(* IEC 61131-3 sources: smart-home/SmartHome/plc (part 3) *)

(* ---- Tn_ReadSensors.st ---- *)
(****************************************************************************
**
** Copyright (C) 2021 Francesco Mandracci
** Contact: https://github.com/fmandracci/smart-home
**
** This file is part of the Smart Home Framework.
**
** Commercial License Usage
** Licensees holding valid commercial licenses may use this file in
** accordance with the terms contained in a written agreement
** between you and the copyright owner.
**
** GNU Lesser General Public License Usage
** Alternatively, this file may be used under the terms of the GNU Lesser
** General Public License version 3 as published by the Free Software
** Foundation and appearing in the file LICENSE included in the
** packaging of this file. Please review the following information to
** ensure the GNU Lesser General Public License version 3 requirements
** will be met: https://www.gnu.org/licenses/lgpl-3.0.html.
**
****************************************************************************)

FUNCTION Tn_ReadSensors
#import "Crosstable.gvl"
#import "Resource1.gvl"
VAR_INPUT
	n  : UINT; (* Tn                     *)
    ES : INT;  (* PLC_Tn_enabled_sensors *)
END_VAR
VAR_IN_OUT
    T1 : INT;  (* PLC_Tn_temperature     *)
    T2 : INT;  (* PLC_Tn_temperature_bis *)
    T3 : INT;  (* PLC_Tn_temperature_ext *)

    H1 : INT;  (* PLC_Tn_humidity        *)
    H2 : INT;  (* PLC_Tn_humidity_bis    *)
    H3 : INT;  (* PLC_Tn_humidity_ext    *)
END_VAR

	(* INPUT: sensors *)
	if PLC_control_type = ControlType_3 or PLC_control_type = ControlType_4 or PLC_control_type = ControlType_15 then
		(* TPAC1007_04_AD Local I/O AI1..3 on RTU3 *)
		if ES >= 1 then
			if NODE_31_STATUS = NODE_NODE_OK then
				SetAnIn_PT100R(PLC_AnInConf_1, PLC_AnIn1Filter);
				T1 := PLC_AnIn_1;
			else
				T1 := TemperatureErrorValue;
			end_if;
			H1 := 0;
		end_if;
		if ES >= 2 then
			if NODE_31_STATUS = NODE_NODE_OK then
				SetAnIn_PT100R(PLC_AnInConf_2, PLC_AnIn2Filter);
				T2 := PLC_AnIn_2;
			else
				T2 := TemperatureErrorValue;
			end_if;
			H2 := 0;
		end_if;
		if ES >= 3 then
			if NODE_31_STATUS = NODE_NODE_OK then
				SetAnIn_PT100R(PLC_AnInConf_3, PLC_AnIn3Filter);
				T3 := PLC_AnIn_3;
			else
				T3 := TemperatureErrorValue;
			end_if;
			H3 := 0;
		end_if;

	elsif (PLC_control_type = ControlType_13 and n <= 3) then
		(* n=1..3 TPAC1007_04_AD Local I/O AI1..3 on RTU3 *)
		if ES >= 1 then
			if NODE_31_STATUS = NODE_NODE_OK then
				case n of
				1:
					SetAnIn_PT100R(PLC_AnInConf_1, PLC_AnIn1Filter);
					T1 := PLC_AnIn_1;
				2:
					SetAnIn_PT100R(PLC_AnInConf_2, PLC_AnIn2Filter);
					T1 := PLC_AnIn_2;
				3:
					SetAnIn_PT100R(PLC_AnInConf_3, PLC_AnIn3Filter);
					T1 := PLC_AnIn_3;
				else ;
				end_case;
			else
				T1 := TemperatureErrorValue;
			end_if;
			H1 := 0;
		end_if;

	elsif PLC_control_type = ControlType_5 or PLC_control_type = ControlType_8 or PLC_control_type = ControlType_12 then
		(* first, second and third (T,H) sensor on RTU3 *)
		if ES <= -1 then
			if NODE_28_STATUS = NODE_NODE_OK then
				T1 := RTU_temperature;
				H1 := RTU_humidity;
			else
				T1 := TemperatureErrorValue;
				H1 := HumidityErrorValue;
			end_if;
		end_if;
		if ES <= -2 then
			if NODE_29_STATUS = NODE_NODE_OK then
				T2 := RTU_temperature_bis;
				H2 := RTU_humidity_bis;
			else
				T2 := TemperatureErrorValue;
				H2 := HumidityErrorValue;
			end_if;
		end_if;
		if ES <= -3 then
			if NODE_30_STATUS = NODE_NODE_OK then
				T3 := RTU_temperature_bis;
				H3 := RTU_humidity_bis;
			else
				T3 := TemperatureErrorValue;
				H3 := HumidityErrorValue;
			end_if;
		end_if;

	elsif PLC_control_type = ControlType_6 then
		(* MPNC 4xAI4 on RTU0 1=C+6 2=B+7 3=A+8 4=base+5, bis,ext varies *)
		if NODE_27_STATUS = NODE_NODE_OK then
			case n of
			1:
				if MPNC_AnInConf_C <> AnIn_MPNCx4_Pt100R then MPNC_AnInConf_C := AnIn_MPNCx4_Pt100R; end_if;
				T1 := MPNC_AnIn_C_3; (* scala *)
				T2 := MPNC_AnIn_C_1; (* lavanderia *)
				T3 := MPNC_AnIn_C_2; (* cantina *)
			2:
				if MPNC_AnInConf_B <> AnIn_MPNCx4_Pt100R then MPNC_AnInConf_B := AnIn_MPNCx4_Pt100R; end_if;
				T1 := MPNC_AnIn_B_3; (* corridoio *)
				T2 := MPNC_AnIn_B_1; (* cucina *)
				T3 := MPNC_AnIn_B_2; (* soggiorno *)
			3:
				if MPNC_AnInConf_A <> AnIn_MPNCx4_Pt100R then MPNC_AnInConf_A := AnIn_MPNCx4_Pt100R; end_if;
				T1 := MPNC_AnIn_A_3; (* sopra sud *)
				T2 := MPNC_AnIn_A_2; (* sopra nord *)
				T3 := MPNC_AnIn_A_1; (* esterna *)
			4:
				if MPNC_AnInConf_1 <> AnIn_MPNC_Pt100R then MPNC_AnInConf_1 := AnIn_MPNC_Pt100R; end_if;
				if MPNC_AnInConf_2 <> AnIn_MPNC_Pt100R then MPNC_AnInConf_2 := AnIn_MPNC_Pt100R; end_if;
				T1 := MPNC_AnIn_1; (* puffer *)
				T2 := MPNC_AnIn_2; (* ritorno radiatori *)
				T3 := 0;
			else ;
			end_case;
		else
			T1 := TemperatureErrorValue;
			T2 := TemperatureErrorValue;
			T3 := TemperatureErrorValue;
		end_if;
		H1 := 0;
		H2 := 0;
		H3 := 0;

	elsif PLC_control_type = ControlType_14 then
		(* MPNC 4xAI4 on RTU0 1=A 2=B 3=C 4=D _1=t _2=t_bis _3=t_ext *)
		if NODE_27_STATUS = NODE_NODE_OK then
			case n of
			1:
				if MPNC_AnInConf_A <> AnIn_MPNCx4_Pt100R then MPNC_AnInConf_A := AnIn_MPNCx4_Pt100R; end_if;
				T1 := MPNC_AnIn_A_1;
				T2 := MPNC_AnIn_A_2;
				T3 := MPNC_AnIn_A_3;
			2:
				if MPNC_AnInConf_B <> AnIn_MPNCx4_Pt100R then MPNC_AnInConf_B := AnIn_MPNCx4_Pt100R; end_if;
				T1 := MPNC_AnIn_B_1;
				T2 := MPNC_AnIn_B_2;
				T3 := MPNC_AnIn_B_3;
			3:
				if MPNC_AnInConf_C <> AnIn_MPNCx4_Pt100R then MPNC_AnInConf_C := AnIn_MPNCx4_Pt100R; end_if;
				T1 := MPNC_AnIn_C_1;
				T2 := MPNC_AnIn_C_2;
				T3 := MPNC_AnIn_C_3;
			4:
				if MPNC_AnInConf_D <> AnIn_MPNCx4_Pt100R then MPNC_AnInConf_D := AnIn_MPNCx4_Pt100R; end_if;
				T1 := MPNC_AnIn_D_1;
				T2 := MPNC_AnIn_D_2;
				T3 := MPNC_AnIn_D_3;
			else ;
			end_case;
		else
			T1 := TemperatureErrorValue;
			T2 := TemperatureErrorValue;
			T3 := TemperatureErrorValue;
		end_if;
		H1 := 0;
		H2 := 0;
		H3 := 0;

	elsif PLC_control_type = ControlType_7 then
		(* n=1..4 MPNE_C AI1..4 on RTU0; n=5,6 T,H on RTU3 *)
		if n <= 4 then
			if ES >= 1 then
				if NODE_13_STATUS = NODE_NODE_OK then
					case n of
					1:
						SetAnIn_PT100R(MPNE_C_AnIn1Conf, MPNE_C_AnIn1Filter);
						T1 := MPNE_C_AnIn_1;
					2:
						SetAnIn_PT100R(MPNE_C_AnIn2Conf, MPNE_C_AnIn2Filter);
						T1 := MPNE_C_AnIn_2;
					3:
						SetAnIn_PT100R(MPNE_C_AnIn3Conf, MPNE_C_AnIn3Filter);
						T1 := MPNE_C_AnIn_3;
					4:
						SetAnIn_PT100R(MPNE_C_AnIn4Conf, MPNE_C_AnIn4Filter);
						T1 := MPNE_C_AnIn_4;
					else ;
					end_case;
				else
					T1 := TemperatureErrorValue;
				end_if;
				H1 := 0;
			end_if;
		elsif (n = 5) and (ES <= -1) then
			if NODE_28_STATUS = NODE_NODE_OK then
				T1 := RTU_temperature;
				H1 := RTU_humidity;
			else
				T1 := TemperatureErrorValue;
				H1 := HumidityErrorValue;
			end_if;
		elsif (n = 6) and (ES <= -1) then
			if NODE_29_STATUS = NODE_NODE_OK then
				T1 := RTU_temperature_bis;
				H1 := RTU_humidity_bis;
			else
				T1 := TemperatureErrorValue;
				H1 := HumidityErrorValue;
			end_if;
		else
			T1 := TemperatureErrorValue;
			H1 := HumidityErrorValue;
		end_if;

	elsif PLC_control_type = ControlType_10 then
		(* MPNE_C AI1.2 on RTU0 *)
		if ES >= 1 then
			if NODE_13_STATUS = NODE_NODE_OK then
				SetAnIn_PT100R(MPNE_C_AnIn1Conf, MPNE_C_AnIn1Filter);
				T1 := MPNE_C_AnIn_1;
			else
				T1 := TemperatureErrorValue;
			end_if;
			H1 := 0;
		end_if;
		if ES >= 2 then
			if NODE_13_STATUS = NODE_NODE_OK then
				SetAnIn_PT100R(MPNE_C_AnIn2Conf, MPNE_C_AnIn2Filter);
				T2 := MPNE_C_AnIn_2;
			else
				T2 := TemperatureErrorValue;
			end_if;
			H2 := 0;
		end_if;

	elsif PLC_control_type = ControlType_11 then
		(* n=1..4: MPNE_C/D AI(1+2) .. (3+4) on RTU0 *)
		case n of
		1:
			SetAnIn_PT100R(MPNE_C_AnIn1Conf, MPNE_C_AnIn1Filter);
			SetAnIn_PT100R(MPNE_C_AnIn2Conf, MPNE_C_AnIn2Filter);
			T1 := MPNE_C_AnIn_1;
			T2 := MPNE_C_AnIn_2;
		2:
			SetAnIn_PT100R(MPNE_C_AnIn3Conf, MPNE_C_AnIn3Filter);
			SetAnIn_PT100R(MPNE_C_AnIn4Conf, MPNE_C_AnIn4Filter);
			T1 := MPNE_C_AnIn_3;
			T2 := MPNE_C_AnIn_4;
		3:
			SetAnIn_PT100R(MPNE_D_AnIn1Conf, MPNE_D_AnIn1Filter);
			SetAnIn_PT100R(MPNE_D_AnIn2Conf, MPNE_D_AnIn2Filter);
			T1 := MPNE_D_AnIn_1;
			T2 := MPNE_D_AnIn_2;
		4:
			SetAnIn_PT100R(MPNE_D_AnIn3Conf, MPNE_D_AnIn3Filter);
			SetAnIn_PT100R(MPNE_D_AnIn4Conf, MPNE_D_AnIn4Filter);
			T1 := MPNE_D_AnIn_3;
			T2 := MPNE_D_AnIn_4;
		else ;
		end_case;

	end_if;

END_FUNCTION

(* ---- Tn_SetDigOut_lamp.st ---- *)
(****************************************************************************
**
** Copyright (C) 2021 Francesco Mandracci
** Contact: https://github.com/fmandracci/smart-home
**
** This file is part of the Smart Home Framework.
**
** Commercial License Usage
** Licensees holding valid commercial licenses may use this file in
** accordance with the terms contained in a written agreement
** between you and the copyright owner.
**
** GNU Lesser General Public License Usage
** Alternatively, this file may be used under the terms of the GNU Lesser
** General Public License version 3 as published by the Free Software
** Foundation and appearing in the file LICENSE included in the
** packaging of this file. Please review the following information to
** ensure the GNU Lesser General Public License version 3 requirements
** will be met: https://www.gnu.org/licenses/lgpl-3.0.html.
**
****************************************************************************)

FUNCTION Tn_SetDigOut_lamp
#import "Crosstable.gvl"
#import "Resource1.gvl"
VAR_INPUT
    x : UINT;
    value : BOOL;
END_VAR

	if PLC_control_type = ControlType_3 or PLC_control_type = ControlType_4 then
		(* TPAC1007_04_AD Local I/O DO1..5 DI7..11 on RTU3 *)
		case x of
		1: if PLC_DigDir_1 <> DigDir_OUT then PLC_DigDir_1 := DigDir_OUT; end_if;
	       if PLC_DigOut_1 <> value      then PLC_DigOut_1 := value; end_if;
		2: if PLC_DigDir_2 <> DigDir_OUT then PLC_DigDir_2 := DigDir_OUT; end_if;
	       if PLC_DigOut_2 <> value      then PLC_DigOut_2 := value; end_if;
		3: if PLC_DigDir_3 <> DigDir_OUT then PLC_DigDir_3 := DigDir_OUT; end_if;
	       if PLC_DigOut_3 <> value      then PLC_DigOut_3 := value; end_if;
		4: if PLC_DigDir_4 <> DigDir_OUT then PLC_DigDir_4 := DigDir_OUT; end_if;
	       if PLC_DigOut_4 <> value      then PLC_DigOut_4 := value; end_if;
		5: if PLC_DigDir_5 <> DigDir_OUT then PLC_DigDir_5 := DigDir_OUT; end_if;
	       if PLC_DigOut_5 <> value      then PLC_DigOut_5 := value; end_if;
 	    else ;
	    end_case;

	elsif PLC_control_type = ControlType_5 or PLC_control_type = ControlType_8 then
		(* Fast I/O FO5..8 FO5..8 on GPIO *)
		case x of
		1: if PLC_FastIO_5 <> value then PLC_FastIO_5 := value; end_if;
		2: if PLC_FastIO_6 <> value then PLC_FastIO_6 := value; end_if;
		3: if PLC_FastIO_7 <> value then PLC_FastIO_7 := value; end_if;
		4: if PLC_FastIO_8 <> value then PLC_FastIO_8 := value; end_if;
 	    else ;
	    end_case;

	else
		; (* no lamps *)
	end_if;

END_FUNCTION

(* ---- Tn_SetDigOut_thermo.st ---- *)
(****************************************************************************
**
** Copyright (C) 2021 Francesco Mandracci
** Contact: https://github.com/fmandracci/smart-home
**
** This file is part of the Smart Home Framework.
**
** Commercial License Usage
** Licensees holding valid commercial licenses may use this file in
** accordance with the terms contained in a written agreement
** between you and the copyright owner.
**
** GNU Lesser General Public License Usage
** Alternatively, this file may be used under the terms of the GNU Lesser
** General Public License version 3 as published by the Free Software
** Foundation and appearing in the file LICENSE included in the
** packaging of this file. Please review the following information to
** ensure the GNU Lesser General Public License version 3 requirements
** will be met: https://www.gnu.org/licenses/lgpl-3.0.html.
**
****************************************************************************)

FUNCTION Tn_SetDigOut_thermo
#import "Crosstable.gvl"
#import "Resource1.gvl"
VAR_INPUT
    n : UINT;
    heating : BOOL;
	only_mantain: BOOL;
	temperature : INT;
	temperature_bis : INT;
END_VAR
VAR_IN_OUT
	last_R : UINT;
END_VAR

	if PLC_control_type = ControlType_3 then
		(* TPAC1007_04_AD DigOut 6 *)
		if NODE_31_STATUS = NODE_NODE_OK then
	    	if PLC_DigDir_6 <> DigDir_OUT then PLC_DigDir_6 := DigDir_OUT; end_if;
			if only_mantain then
				; (* do nothing *)
			else
		        if PLC_DigOut_6 <> HEATING then PLC_DigOut_6 := HEATING; end_if;
		    end_if;
	    end_if;

	elsif PLC_control_type = ControlType_4 or PLC_control_type = ControlType_5 or PLC_control_type = ControlType_8 then
		(* ARQ01 relè *)
		if NODE_10_STATUS = NODE_NODE_OK then
		    if only_mantain then
				; (* do nothing *)
			else
		        if ARQ_Rele <> HEATING then ARQ_Rele := HEATING; end_if;
			end_if;
		end_if;

	elsif PLC_control_type = ControlType_7 then
		(* n=1..4: MPNE_C DigOut 1..4 *)
		if NODE_13_STATUS = NODE_NODE_OK then
			if only_mantain then
				; (* do nothing *)
			else
	    		case n of
				1:
			    	if MPNE_C_DigDir_1 <> DigDir_OUT then MPNE_C_DigDir_1 := DigDir_OUT; end_if;
			        if MPNE_C_DigOut_1 <> HEATING    then MPNE_C_DigOut_1 := HEATING   ; end_if;
				2:
			    	if MPNE_C_DigDir_2 <> DigDir_OUT then MPNE_C_DigDir_2 := DigDir_OUT; end_if;
			        if MPNE_C_DigOut_2 <> HEATING    then MPNE_C_DigOut_2 := HEATING   ; end_if;
				3:
			    	if MPNE_C_DigDir_3 <> DigDir_OUT then MPNE_C_DigDir_3 := DigDir_OUT; end_if;
			        if MPNE_C_DigOut_3 <> HEATING    then MPNE_C_DigOut_3 := HEATING   ; end_if;
				4:
			    	if MPNE_C_DigDir_4 <> DigDir_OUT then MPNE_C_DigDir_4 := DigDir_OUT; end_if;
			        if MPNE_C_DigOut_4 <> HEATING    then MPNE_C_DigOut_4 := HEATING   ; end_if;
				5:
			    	if MPNE_C_DigDir_5 <> DigDir_OUT then MPNE_C_DigDir_5 := DigDir_OUT; end_if;
			        if MPNE_C_DigOut_5 <> HEATING    then MPNE_C_DigOut_5 := HEATING   ; end_if;
				6:
			    	if MPNE_C_DigDir_6 <> DigDir_OUT then MPNE_C_DigDir_6 := DigDir_OUT; end_if;
			        if MPNE_C_DigOut_6 <> HEATING    then MPNE_C_DigOut_6 := HEATING   ; end_if;
				else ;
				end_case;
			end_if;
		end_if;

	elsif PLC_control_type = ControlType_10 then
		(* MPNE_C DigOut 1 *)
		if NODE_13_STATUS = NODE_NODE_OK then
	    	if MPNE_C_DigDir_1 <> DigDir_OUT then MPNE_C_DigDir_1 := DigDir_OUT; end_if;

			if only_mantain then
				; (* do nothing *)
			else
		        if heating then (* see also Tn_OverHeat() *)
			    	if not MPNE_C_DigOut_1 then MPNE_C_DigOut_1 := true; end_if;
				else
			    	if MPNE_C_DigOut_1 then MPNE_C_DigOut_1 := false; end_if;
				end_if;
			end_if;
		end_if;

	elsif PLC_control_type = ControlType_11 then
		(* i=1..4: MPNE_C/_D DigOut 1.2 *)
		if n <= 2 then
			if NODE_13_STATUS = NODE_NODE_OK then
				if only_mantain then
					; (* do nothing *)
				else
					case n of
					1:
				    	if MPNE_C_DigDir_1 <> DigDir_OUT then MPNE_C_DigDir_1 := DigDir_OUT; end_if;
						if only_mantain then
							; (* do nothing *)
						else
					        if heating then (* see also Tn_OverHeat() *)
						    	if not MPNE_C_DigOut_1 then MPNE_C_DigOut_1 := true; end_if;
							else
						    	if MPNE_C_DigOut_1 then MPNE_C_DigOut_1 := false; end_if;
							end_if;
						end_if;
					2:
				    	if MPNE_C_DigDir_2 <> DigDir_OUT then MPNE_C_DigDir_2 := DigDir_OUT; end_if;
						if only_mantain then
							; (* do nothing *)
						else
					        if heating then (* see also Tn_OverHeat() *)
						    	if not MPNE_C_DigOut_2 then MPNE_C_DigOut_2 := true; end_if;
							else
						    	if MPNE_C_DigOut_2 then MPNE_C_DigOut_2 := false; end_if;
							end_if;
						end_if;
					else ;
					end_case;
				end_if;
			end_if;
		else
			if NODE_14_STATUS = NODE_NODE_OK then
				if only_mantain then
					; (* do nothing *)
				else
					case n of
					3:
				    	if MPNE_D_DigDir_1 <> DigDir_OUT then MPNE_D_DigDir_1 := DigDir_OUT; end_if;
						if only_mantain then
							; (* do nothing *)
						else
					        if heating then (* see also Tn_OverHeat() *)
						    	if not MPNE_D_DigOut_1 then MPNE_D_DigOut_1 := true; end_if;
							else
						    	if MPNE_D_DigOut_1 then MPNE_D_DigOut_1 := false; end_if;
							end_if;
						end_if;
					4:
				    	if MPNE_D_DigDir_2 <> DigDir_OUT then MPNE_D_DigDir_2 := DigDir_OUT; end_if;
						if only_mantain then
							; (* do nothing *)
						else
					        if heating then (* see also Tn_OverHeat() *)
						    	if not MPNE_D_DigOut_2 then MPNE_D_DigOut_2 := true; end_if;
							else
						    	if MPNE_D_DigOut_2 then MPNE_D_DigOut_2 := false; end_if;
							end_if;
						end_if;
					else ;
					end_case;
				end_if;
			end_if;
		end_if;

	elsif PLC_control_type = ControlType_12 then
		(* FastI/O FO 8 *)
        if only_mantain then
			; (* do nothing *)
		else
	        if PLC_FastIO_8 <> HEATING then PLC_FastIO_8 := HEATING; end_if;
		end_if;

	elsif PLC_control_type = ControlType_13 then
		(* n=1..4: TPAC1007_04_AD DigOut_1..4 *)
		if NODE_31_STATUS = NODE_NODE_OK then
			if only_mantain then
				; (* do nothing *)
			else
		        case n of
				1:
			    	if PLC_DigDir_1 <> DigDir_OUT then PLC_DigDir_1 := DigDir_OUT; end_if;
			        if PLC_DigOut_1 <> HEATING    then PLC_DigOut_1 := HEATING   ; end_if;
				2:
			    	if PLC_DigDir_2 <> DigDir_OUT then PLC_DigDir_2 := DigDir_OUT; end_if;
			        if PLC_DigOut_2 <> HEATING    then PLC_DigOut_2 := HEATING   ; end_if;
				3:
			    	if PLC_DigDir_3 <> DigDir_OUT then PLC_DigDir_3 := DigDir_OUT; end_if;
			        if PLC_DigOut_3 <> HEATING    then PLC_DigOut_3 := HEATING   ; end_if;
				4:
			    	if PLC_DigDir_4 <> DigDir_OUT then PLC_DigDir_4 := DigDir_OUT; end_if;
			        if PLC_DigOut_4 <> HEATING    then PLC_DigOut_4 := HEATING   ; end_if;
				else ;
				end_case;
			end_if;
		end_if;

	elsif PLC_control_type = ControlType_6 then
		(* MPNC 4xAI4 on RTU0 1=C+6 2=B+7 3=A+8 4=base+5, bis,ext varies *)
		if NODE_27_STATUS = NODE_NODE_OK then
			if only_mantain then
				; (* do nothing *)
			else
		        case n of
				1:
			    	if MPNC_DigDir_6 <> DigDir_OUT then MPNC_DigDir_6 := DigDir_OUT; end_if;
			        if MPNC_DigOut_6 <> HEATING    then MPNC_DigOut_6 := HEATING   ; end_if;
				2:
			    	if MPNC_DigDir_7 <> DigDir_OUT then MPNC_DigDir_7 := DigDir_OUT; end_if;
			        if MPNC_DigOut_7 <> HEATING    then MPNC_DigOut_7 := HEATING   ; end_if;
				3:
			    	if MPNC_DigDir_8 <> DigDir_OUT then MPNC_DigDir_8 := DigDir_OUT; end_if;
			        if MPNC_DigOut_8 <> HEATING    then MPNC_DigOut_8 := HEATING   ; end_if;
				4:
			    	if MPNC_DigDir_5 <> DigDir_OUT then MPNC_DigDir_5 := DigDir_OUT; end_if;
			        if MPNC_DigOut_5 <> HEATING    then MPNC_DigOut_5 := HEATING   ; end_if;
				else ;
				end_case;
			end_if;
		end_if;

	elsif PLC_control_type = ControlType_14 then
		(* n=1..4: MPNC base DigOut_1..4 *)
		if NODE_27_STATUS = NODE_NODE_OK then
			if only_mantain then
				; (* do nothing *)
			else
		        case n of
				1:
			    	if MPNC_DigDir_1 <> DigDir_OUT then MPNC_DigDir_1 := DigDir_OUT; end_if;
			        if MPNC_DigOut_1 <> HEATING    then MPNC_DigOut_1 := HEATING   ; end_if;
				2:
			    	if MPNC_DigDir_2 <> DigDir_OUT then MPNC_DigDir_2 := DigDir_OUT; end_if;
			        if MPNC_DigOut_2 <> HEATING    then MPNC_DigOut_2 := HEATING   ; end_if;
				3:
			    	if MPNC_DigDir_3 <> DigDir_OUT then MPNC_DigDir_3 := DigDir_OUT; end_if;
			        if MPNC_DigOut_3 <> HEATING    then MPNC_DigOut_3 := HEATING   ; end_if;
				4:
			    	if MPNC_DigDir_4 <> DigDir_OUT then MPNC_DigDir_4 := DigDir_OUT; end_if;
			        if MPNC_DigOut_4 <> HEATING    then MPNC_DigOut_4 := HEATING   ; end_if;
				else ;
				end_case;
		    end_if;
	    end_if;

	elsif PLC_control_type = ControlType_15 then
		(* TPAC1007_04_AD DigOut_8 *)
		if NODE_31_STATUS = NODE_NODE_OK then
	    	if PLC_DigDir_8 <> DigDir_OUT then PLC_DigDir_8 := DigDir_OUT; end_if;
	        if only_mantain then
				; (* do nothing *)
			else
		        if PLC_DigOut_8 <> HEATING then PLC_DigOut_8 := HEATING; end_if;
			end_if;
	    end_if;

	end_if;

END_FUNCTION

(* ---- Tn_Watchdog.st ---- *)
(****************************************************************************
**
** Copyright (C) 2021 Francesco Mandracci
** Contact: https://github.com/fmandracci/smart-home
**
** This file is part of the Smart Home Framework.
**
** Commercial License Usage
** Licensees holding valid commercial licenses may use this file in
** accordance with the terms contained in a written agreement
** between you and the copyright owner.
**
** GNU Lesser General Public License Usage
** Alternatively, this file may be used under the terms of the GNU Lesser
** General Public License version 3 as published by the Free Software
** Foundation and appearing in the file LICENSE included in the
** packaging of this file. Please review the following information to
** ensure the GNU Lesser General Public License version 3 requirements
** will be met: https://www.gnu.org/licenses/lgpl-3.0.html.
**
****************************************************************************)

FUNCTION Tn_Watchdog
#import "Crosstable.gvl"
#import "Resource1.gvl"

	if (PLC_control_type = ControlType_4) or (PLC_control_type = ControlType_5) or (PLC_control_type = ControlType_8) then
		if ARQ_Watchdog <> WatchDogTimeout_s and NODE_10_STATUS = NODE_NODE_OK then
			ARQ_Watchdog := WatchDogTimeout_s;
		end_if;
	end_if;

END_FUNCTION

(* ---- FilteredSensors.st ---- *)
(****************************************************************************
**
** Copyright (C) 2021 Francesco Mandracci
** Contact: https://github.com/fmandracci/smart-home
**
** This file is part of the Smart Home Framework.
**
** Commercial License Usage
** Licensees holding valid commercial licenses may use this file in
** accordance with the terms contained in a written agreement
** between you and the copyright owner.
**
** GNU Lesser General Public License Usage
** Alternatively, this file may be used under the terms of the GNU Lesser
** General Public License version 3 as published by the Free Software
** Foundation and appearing in the file LICENSE included in the
** packaging of this file. Please review the following information to
** ensure the GNU Lesser General Public License version 3 requirements
** will be met: https://www.gnu.org/licenses/lgpl-3.0.html.
**
****************************************************************************)

FUNCTION_BLOCK FilteredSensors
#import "Crosstable.gvl"
#import "Resource1.gvl"
VAR_INPUT
	n  : UINT; (* Tn                     *)
    ES : INT;  (* PLC_Tn_enabled_sensors *)
END_VAR
VAR_IN_OUT
    T1 : INT;  (* PLC_Tn_temperature     *)
    T2 : INT;  (* PLC_Tn_temperature_bis *)
    T3 : INT;  (* PLC_Tn_temperature_ext *)

    H1 : INT;  (* PLC_Tn_humidity        *)
    H2 : INT;  (* PLC_Tn_humidity_bis    *)
    H3 : INT;  (* PLC_Tn_humidity_ext    *)
END_VAR
VAR
    T1_value : INT := TemperatureErrorValue;
    T2_value : INT := TemperatureErrorValue;
    T3_value : INT := TemperatureErrorValue;
	i : INT;
	s : INT;
	m : INT;
	first_time : BOOL := true;
	T1_array : array [1 .. RollingAverageSize] of INT;
	T2_array : array [1 .. RollingAverageSize] of INT;
	T3_array : array [1 .. RollingAverageSize] of INT;
END_VAR

	if first_time then
		first_time := false;
		for i := 1 to RollingAverageSize by 1 do
			T1_array[i] := TemperatureErrorValue;
			T2_array[i] := TemperatureErrorValue;
			T3_array[i] := TemperatureErrorValue;
		end_for;
	end_if;

    Tn_ReadSensors(n, ES, T1_value, T2_value, T3_value, H1, H2, H3);

	if (abs(ES) >= 1) and (T1_value <> TemperatureErrorValue) then
		s := 0;
		for i := 1 to (RollingAverageSize - 1) by 1 do
			T1_array[i] := T1_array[i + 1];
			s := s + T1_array[i];
		end_for;
		T1_array[RollingAverageSize] := T1_value;
		s := s + T1_value;
		m := s / RollingAverageSize;
		if (s mod RollingAverageSize) >= HalfRollingAverageSize then
			m := m + 1;
		end_if;
		if abs(T1_value - m) <= RollingAverageMaxDeltaT then
			T1 := m;
		else
			for i := 1 to RollingAverageSize by 1 do
				T1_array[i] := T1_value;
			end_for;
			T1 := T1_value;
		end_if;
	else
		T1 := TemperatureErrorValue;
	end_if;

	if (abs(ES) >= 2) and (T2_value <> TemperatureErrorValue) then
		s := 0;
		for i := 1 to (RollingAverageSize - 1) by 1 do
			T2_array[i] := T2_array[i + 1];
			s := s + T2_array[i];
		end_for;
		T2_array[RollingAverageSize] := T2_value;
		s := s + T2_value;
		m := s / RollingAverageSize;
		if (s mod RollingAverageSize) >= HalfRollingAverageSize then
			m := m + 1;
		end_if;
		if abs(T2_value - m) <= RollingAverageMaxDeltaT then
			T2 := m;
		else
			for i := 1 to RollingAverageSize by 1 do
				T2_array[i] := T2_value;
			end_for;
			T2 := T2_value;
		end_if;
	else
		T2 := TemperatureErrorValue;
	end_if;

	if (abs(ES) >= 3) and (T3_value <> TemperatureErrorValue) then
		s := 0;
		for i := 1 to (RollingAverageSize - 1) by 1 do
			T3_array[i] := T3_array[i + 1];
			s := s + T3_array[i];
		end_for;
		T3_array[RollingAverageSize] := T3_value;
		s := s + T3_value;
		m := s / RollingAverageSize;
		if (s mod RollingAverageSize) >= HalfRollingAverageSize then
			m := m + 1;
		end_if;
		if abs(T3_value - m) <= RollingAverageMaxDeltaT then
			T3 := m;
		else
			for i := 1 to RollingAverageSize by 1 do
				T3_array[i] := T3_value;
			end_for;
			T3 := T3_value;
		end_if;
	else
		T3 := TemperatureErrorValue;
	end_if;

END_FUNCTION_BLOCK

(* ---- LampImpulse.st ---- *)
(****************************************************************************
**
** Copyright (C) 2021 Francesco Mandracci
** Contact: https://github.com/fmandracci/smart-home
**
** This file is part of the Smart Home Framework.
**
** Commercial License Usage
** Licensees holding valid commercial licenses may use this file in
** accordance with the terms contained in a written agreement
** between you and the copyright owner.
**
** GNU Lesser General Public License Usage
** Alternatively, this file may be used under the terms of the GNU Lesser
** General Public License version 3 as published by the Free Software
** Foundation and appearing in the file LICENSE included in the
** packaging of this file. Please review the following information to
** ensure the GNU Lesser General Public License version 3 requirements
** will be met: https://www.gnu.org/licenses/lgpl-3.0.html.
**
****************************************************************************)

FUNCTION_BLOCK LampImpulse
VAR_INPUT
    x  : UINT;
END_VAR
VAR_IN_OUT
    PLC_Tn_lamp_x : BOOL;
    SRV_Tn_lamp_x : BOOL;
    PLC_Tn_lamp_feedback_x : BOOL;
END_VAR
VAR
	active : BOOL := false;
END_VAR;

	if active then
        Tn_SetDigOut_lamp(x, false);
		PLC_Tn_lamp_x := false;
        SRV_Tn_lamp_x := false;
		active := false;
    else
	    if PLC_Tn_lamp_x or SRV_Tn_lamp_x then
	        Tn_SetDigOut_lamp(x, true);
			active := true;
		end_if;
	end_if;

    PLC_Tn_lamp_feedback_x := Tn_GetDigIn_lamp(x);

END_FUNCTION_BLOCK

(* ---- Thermostat.st ---- *)
(****************************************************************************
**
** Copyright (C) 2021 Francesco Mandracci
** Contact: https://github.com/fmandracci/smart-home
**
** This file is part of the Smart Home Framework.
**
** Commercial License Usage
** Licensees holding valid commercial licenses may use this file in
** accordance with the terms contained in a written agreement
** between you and the copyright owner.
**
** GNU Lesser General Public License Usage
** Alternatively, this file may be used under the terms of the GNU Lesser
** General Public License version 3 as published by the Free Software
** Foundation and appearing in the file LICENSE included in the
** packaging of this file. Please review the following information to
** ensure the GNU Lesser General Public License version 3 requirements
** will be met: https://www.gnu.org/licenses/lgpl-3.0.html.
**
****************************************************************************)

FUNCTION_BLOCK Thermostat
#import "Crosstable.gvl"
#import "Resource1.gvl"
VAR_INPUT
	N : UINT;   (* Tn                             *)
    ES : INT;   (* PLC_Tn_enabled_sensors         *)
	NT : BOOL;  (* PLC_Tn_nighttime               *)

    T_1 : INT;  (* PLC_Tn_temperature             *)
    T_2 : INT;  (* PLC_Tn_temperature_bis         *)

    H_1 : INT;  (* PLC_Tn_humidity                *)
    H_2 : INT;  (* PLC_Tn_humidity_bis            *)

	M_W : UINT; (* PLC_Tn_max_request_W           *)
	A_W : UINT; (* PLC_EP_Tn_assigned_W           *)
END_VAR
VAR_IN_OUT
	PRW : UINT; (* PLC_Tn_requested_W             *)
	SRW : UINT; (* SRV_Tn_requested_W             *)

    TSP : INT;  (* PLC_Tn_temperature_setpoint    *)
    TSPN: INT;  (* PLC_Tn_temperature_setpoint_nt *)

    HSP : INT;  (* PLC_Tn_humidity_setpoint       *)
    HSPN: INT;  (* PLC_Tn_humidity_setpoint_nt    *)

    PLC_STATUS  : INT ; (* PLC_Tn_heating_status  *)
    PLC_TIMER   : INT ; (* PLC_Tn_heating_timer   *)
    PLC_HEATING : BOOL; (* PLC_Tn_heating         *)

    SRV_STATUS  : INT ; (* SRV_Tn_heating_status  *)
    SRV_TIMER   : INT ; (* SRV_Tn_heating_timer   *)
    SRV_HEATING : BOOL; (* SRV_Tn_heating         *)

    DH  : UDINT ; (* PLC_Tn_daily_heating_s       *)
    MH  : UDINT ; (* PLC_Tn_monthly_heating_s     *)
END_VAR
VAR
	HEATING : BOOL;
	TIMER : INT;
	STATUS : INT;
	A_TSP : INT; (* actual temperature setpoint, changed by ECONOMY, COMFORT, BOOST and nightime *)
	A_HSP : INT; (* actual humidity setpoint, NOT changed by ECONOMY, COMFORT, BOOST and nightime *)
	last_R : UINT := 0;
END_VAR;

	STATUS := PLC_STATUS;
	TIMER := PLC_TIMER;
	HEATING := PLC_HEATING;

	(* ----------------- 1/4 common ----------------- *)

	(* check nightime and limits *)
	if NT then
		A_TSP := Tn_CheckSetpoint_T(TSPN);
		A_HSP := Tn_CheckSetpoint_H(HSPN);
		(* NB: may change setpoints <---------------- *)
		if TSPN <> A_TSP then TSPN := A_TSP; end_if;
		if HSPN <> A_HSP then HSPN := A_HSP; end_if;
	else
		A_TSP := Tn_CheckSetpoint_T(TSP);
		A_HSP := Tn_CheckSetpoint_H(HSP);
		(* NB: may change setpoints <---------------- *)
		if TSP <> A_TSP then TSP := A_TSP; end_if;
		if HSP <> A_HSP then HSP := A_HSP; end_if;
	end_if;

	(* check timer *)
	if STATUS > HEATING_AUTO then
		if TIMER > 0 then
		    TIMER := TIMER - 1;
		else
			STATUS := HEATING_AUTO;
			TIMER := 0;
		end_if;
	end_if;

	(* check special states *)
	case STATUS of
	HEATING_AUTO:
		A_TSP := A_TSP;
	HEATING_ECONOMY:
		A_TSP := A_TSP - 20; (* -2°C*) (* ex: -10% A_TSP - (A_TSP * 100) / 10; *)
	HEATING_COMFORT:
		A_TSP := A_TSP + 20; (* +2°C*) (* ex: +10% A_TSP + (A_TSP * 100) / 10; *)
	HEATING_BOOST:
		A_TSP := TemperatureSetPoint_max;
	else
		;
	end_case;

	(* check limits after changes *)
	A_TSP := Tn_CheckSetpoint_T(A_TSP);
	A_HSP := Tn_CheckSetpoint_H(A_HSP);

	(* ----------------- 2/4 common control ----------------- *)

	if PLC_control_type = ControlType_0 or PLC_control_type = ControlType_1  or PLC_control_type = ControlType_2 then
		(* no thermostat *)
	    HEATING := false;

	elsif ES = 0 or (abs(ES) >= 1 and T_1 = TemperatureErrorValue) or (abs(ES) >= 2 and T_2 = TemperatureErrorValue) then
		(* sensor read error *)
	    HEATING := false;

	elsif (ES <= -1 and H_1 = HumidityErrorValue) or (ES <= -2 and H_2 = HumidityErrorValue) then
		(* sensor read error *)
	    HEATING := false;

	elsif (PLC_control_type = ControlType_6 and n = 4) or (PLC_control_type = ControlType_15 and n = 1) then
		(* differential thermostat (puffer) *)
		if PLC_UPTIME_s <= 25 then
			(* waiting for sensors settling *)
			HEATING := false;
		elsif STATUS >= HEATING_AUTO then
			(* heating enabled *)
			if HEATING then
				(* heating was ON *)
				if T_1 < (T_2 - TemperatureHysteresis) then
					(* puffer is colder than thermo water *)
					HEATING := false;
				end_if;
			else
				(* heating was off *)
				if  T_1 >= (T_2 + TemperatureHysteresis) then
					(* puffer is warmer than thermo water *)
					HEATING := true;
				end_if;
			end_if;
		else
			HEATING := false;
			TIMER := 0;
		end_if;

	else
		(* standard thermostat *)
		if PLC_UPTIME_s <= 25 then
			(* waiting for sensors settling *)
			HEATING := false;
		elsif STATUS >= HEATING_AUTO then
			(* heating enabled *)
			if HEATING then
				(* heating was ON *)
				if (ES <= -2)   and ( T_1 >= (A_TSP + TemperatureHysteresis) AND T_2 >= (A_TSP + TemperatureHysteresis) AND H_1 <= (A_HSP - HumidityHysteresis) AND H_2 <= (A_HSP - HumidityHysteresis) ) then
					(* two T,H sensors *)
					HEATING := false;
				elsif (ES = -1) and ( T_1 >= (A_TSP + TemperatureHysteresis)                                            AND H_1 <= (A_HSP - HumidityHysteresis)                                     ) then
					(* one T,H sensor *)
					HEATING := false;
				elsif (ES = 0) then
					(* nothing *)
					HEATING := false;
				elsif (ES = 1)  and ( T_1 >= (A_TSP + TemperatureHysteresis) ) then
					(* one Pt100 *)
					HEATING := false;
				elsif (ES >= 2) and ( T_1 >= (A_TSP + TemperatureHysteresis) AND T_2 >= (A_TSP + TemperatureHysteresis)  ) then
					(* two Pt100s *)
					HEATING := false;
				end_if;
			else
				(* heating was off *)
				if (ES <= -2)   and ( T_1 <= (A_TSP - TemperatureHysteresis) OR T_2 <= (A_TSP - TemperatureHysteresis) OR H_1 >= (A_HSP + HumidityHysteresis) OR H_2 >= (A_HSP + HumidityHysteresis) ) then
					(* two T,H sensors *)
					HEATING := true;
				elsif (ES = -1) and ( T_1 <= (A_TSP - TemperatureHysteresis)                                           OR H_1 >= (A_HSP + HumidityHysteresis)                                    ) then
					(* one T,H sensor *)
					HEATING := true;
				elsif (ES = 0) then
					(* nothing *)
					HEATING := false;
				elsif (ES = 1)  and ( T_1 <= (A_TSP - TemperatureHysteresis) ) then
					(* one Pt100 *)
					HEATING := true;
				elsif (ES >= 2) and ( T_1 <= (A_TSP - TemperatureHysteresis) OR T_2 <= (A_TSP - TemperatureHysteresis) ) then
					(* two Pt100s *)
					HEATING := true;
				end_if;
			end_if;
		else
			HEATING := false;
			TIMER := 0;
		end_if;

	end_if;

	(* ----------------- 3/4 specific control and action ----------------- *)

	if HEATING and Tn_OverHeat(n, T_1, T_2) then
		HEATING := false;
	end_if;

	if M_W = 0 or not PLC_EP_exists then
		(* no load balancing *)
	   	Tn_SetDigOut_thermo(n, HEATING, false, T_1, T_2, last_R);
		if PRW <> 0 then
			PRW := 0; (* PLC_Tn_requested_W := 0 *)
		end_if;

	elsif not PLC_EP_isOK then
		(* safe state *)
		HEATING := false;
	   	Tn_SetDigOut_thermo(n, false, false, T_1, T_2, last_R);

	elsif not HEATING then
		(* simply power off *)
	   	Tn_SetDigOut_thermo(n, false, false, T_1, T_2, last_R);
		PRW := 0; (* PLC_Tn_requested_W *)
		if SRW <> 0 then SRW := 0; end_if; (* SRV_Tn_requested_W *)

	else

		case PLC_EP_tic_in_tac of

	    0: (* request time *)
			PRW := M_W; (* PLC_Tn_requested_W := PLC_Tn_max_request_W *)
			if SRW <> M_W then
				SRW := M_W; (* SRV_Tn_requested_W := PLC_Tn_max_request_W *)
			end_if;
			(* wait, only maintain the current status *)
			Tn_SetDigOut_thermo(n, false, true, T_1, T_2, last_R);

		1: (* transmission time *)
			(* wait, only maintain the current status *)
			Tn_SetDigOut_thermo(n, false, true, T_1, T_2, last_R);

		Decision_TicInTac: (* decision time *)
			(* wait, only maintain the current status *)
			Tn_SetDigOut_thermo(n, false, true, T_1, T_2, last_R);

		3: (* transmission time *)
			(* wait, only maintain the current status *)
			Tn_SetDigOut_thermo(n, false, true, T_1, T_2, last_R);

		4:	(* power off time *)
			if A_W >= M_W then (* PLC_EP_Tn_assigned_W >= PLC_Tn_max_request_W *)
				(* wait, only maintain the current status *)
				Tn_SetDigOut_thermo(n, false, true, T_1, T_2, last_R);
			else
				(* power off *)
			   	Tn_SetDigOut_thermo(n, false, false, T_1, T_2, last_R);
			end_if;

		5:
			(* action time *)
			if A_W >= M_W then (* PLC_EP_Tn_assigned_W >= PLC_Tn_max_request_W *)
			   	Tn_SetDigOut_thermo(n, true, false, T_1, T_2, last_R);
			else
			   	Tn_SetDigOut_thermo(n, false, false, T_1, T_2, last_R);
			end_if;

		6:
			(* action time bis *)
			if A_W >= M_W then (* PLC_EP_Tn_assigned_W >= PLC_Tn_max_request_W *)
			   	Tn_SetDigOut_thermo(n, true, false, T_1, T_2, last_R);
			else
			   	Tn_SetDigOut_thermo(n, false, false, T_1, T_2, last_R);
			end_if;

		end_case;

	end_if;

	(* ----------------- 4/4 update ----------------- *)

	if PLC_STATUS <> STATUS then
		PLC_STATUS := STATUS;
		SRV_STATUS := STATUS;
	end_if;
	if PLC_TIMER <> TIMER then
		PLC_TIMER := TIMER;
		SRV_TIMER := TIMER;
	end_if;
	if PLC_HEATING <> HEATING then
		PLC_HEATING := HEATING;
		SRV_HEATING := HEATING;
	end_if;

	if (PLC_Hours = 0) and (PLC_Minutes = 0) and (PLC_Seconds = 0) then
		DH := 0;
		if PLC_Day = 1 then
			MH := 0;
		end_if;
	elsif HEATING then
		DH := DH + 1;
		MH := MH + 1;
	end_if;

END_FUNCTION_BLOCK

(* ---- Alarms.st ---- *)
(****************************************************************************
**
** Copyright (C) 2021 Francesco Mandracci
** Contact: https://github.com/fmandracci/smart-home
**
** This file is part of the Smart Home Framework.
**
** Commercial License Usage
** Licensees holding valid commercial licenses may use this file in
** accordance with the terms contained in a written agreement
** between you and the copyright owner.
**
** GNU Lesser General Public License Usage
** Alternatively, this file may be used under the terms of the GNU Lesser
** General Public License version 3 as published by the Free Software
** Foundation and appearing in the file LICENSE included in the
** packaging of this file. Please review the following information to
** ensure the GNU Lesser General Public License version 3 requirements
** will be met: https://www.gnu.org/licenses/lgpl-3.0.html.
**
****************************************************************************)

PROGRAM Alarms
#import "Crosstable.gvl"
#import "Resource1.gvl"
VAR

END_VAR

;

END_PROGRAM

(* ---- BA_main.st ---- *)
(****************************************************************************
**
** Copyright (C) 2021 Francesco Mandracci
** Contact: https://github.com/fmandracci/smart-home
**
** This file is part of the Smart Home Framework.
**
** Commercial License Usage
** Licensees holding valid commercial licenses may use this file in
** accordance with the terms contained in a written agreement
** between you and the copyright owner.
**
** GNU Lesser General Public License Usage
** Alternatively, this file may be used under the terms of the GNU Lesser
** General Public License version 3 as published by the Free Software
** Foundation and appearing in the file LICENSE included in the
** packaging of this file. Please review the following information to
** ensure the GNU Lesser General Public License version 3 requirements
** will be met: https://www.gnu.org/licenses/lgpl-3.0.html.
**
****************************************************************************)

PROGRAM BA_main
#import "Crosstable.gvl"
#import "Resource1.gvl"
VAR
	substatus : UINT := 0;
	timer : TON;
	NEXT_STATUS : UINT := 0;
	NEXT_INDEX : UINT := 0;
END_VAR;

    if not PLC_Iam_BA then
		return;
    end_if;
	if PLC_BA_just_started then
		PLC_BA_just_started := false;
		timer(IN := FALSE);
		substatus := 0;
	end_if;

	BA_Watchdog();

	NEXT_STATUS := PLC_BA_status;
	NEXT_INDEX := PLC_BA_config_index;

	case substatus of

	0: (* ----- recover config  ------------------------------------------- *)

		case PLC_BA_status of
		ALARM_STATUS_ZERO:
			NEXT_INDEX := ALARM_INDEX_NOTHING;
			NEXT_STATUS := ALARM_STATUS_OFF;
		ALARM_STATUS_OFF:
			NEXT_INDEX := ALARM_INDEX_NOTHING;
		ALARM_STATUS_ARMED:
			;
		ALARM_STATUS_ENABLED:
			;
		ALARM_STATUS_RINGING:
			;
		ALARM_STATUS_MUTED:
			;
		ALARM_STATUS_TESTING:
			;
		else
			NEXT_INDEX := ALARM_INDEX_NOTHING;
			NEXT_STATUS := ALARM_STATUS_OFF;
		end_case;

		BA_WriteConfig(NEXT_INDEX, PLC_BA_config_index, PLC_BA_config_mask);
	    PLC_BA_command := ALARM_COMMAND_NONE;
		substatus := 1;

	1: (* ----- waiting config after write -------------------------------- *)

		timer(IN := TRUE, PT := ControlPeriod);
		if timer.Q then
			timer(IN := FALSE);
			substatus := 2;
		end_if;

	2: (* ----- read sensors ---------------------------------------------- *)

		BA_ReadSensors();
		substatus := 3;

	3: (* ----- check sensors --------------------------------------------- *)

		case PLC_BA_status of

		ALARM_STATUS_ZERO:
			BA_ClearOKs();
			NEXT_INDEX := ALARM_INDEX_NOTHING;
			NEXT_STATUS := ALARM_STATUS_OFF;
			BA_WriteConfig(NEXT_INDEX, PLC_BA_config_index, PLC_BA_config_mask);
			substatus := 1;

		ALARM_STATUS_OFF:
			BA_ClearOKs();
			if PLC_BA_command = ALARM_COMMAND_DAYTIME then
				NEXT_STATUS := ALARM_STATUS_ARMED;
				NEXT_INDEX := ALARM_INDEX_DAYTIME;
				BA_WriteConfig(NEXT_INDEX, PLC_BA_config_index, PLC_BA_config_mask);
				substatus := 1;
			elsif PLC_BA_command = ALARM_COMMAND_NIGHTTIME then
				NEXT_STATUS := ALARM_STATUS_ARMED;
				NEXT_INDEX := ALARM_INDEX_NIGHTTIME;
				BA_WriteConfig(NEXT_INDEX, PLC_BA_config_index, PLC_BA_config_mask);
				substatus := 1;
			elsif PLC_BA_command = ALARM_COMMAND_EVERYTHING then
				NEXT_STATUS := ALARM_STATUS_ARMED;
				NEXT_INDEX := ALARM_INDEX_EVERYTHING;
				BA_WriteConfig(NEXT_INDEX, PLC_BA_config_index, PLC_BA_config_mask);
				substatus := 1;
			elsif PLC_BA_command = ALARM_COMMAND_TEST then
				NEXT_STATUS := ALARM_STATUS_TESTING;
				(* NEXT_INDEX := ALARM_INDEX_NOTHING; *)
			 	(* no BA_WriteConfig(NEXT_INDEX, PLC_BA_config_index, PLC_BA_config_mask);     *)
				substatus := 2;
			else
				substatus := 2;
			end_if;

		ALARM_STATUS_ARMED:
			if PLC_BA_command = ALARM_COMMAND_DAYTIME then
				NEXT_INDEX := ALARM_INDEX_DAYTIME;
				BA_WriteConfig(NEXT_INDEX, PLC_BA_config_index, PLC_BA_config_mask);
				substatus := 1;
			elsif PLC_BA_command = ALARM_COMMAND_NIGHTTIME then
				NEXT_INDEX := ALARM_INDEX_NIGHTTIME;
				BA_WriteConfig(NEXT_INDEX, PLC_BA_config_index, PLC_BA_config_mask);
				substatus := 1;
			elsif PLC_BA_command = ALARM_COMMAND_EVERYTHING then
				NEXT_INDEX := ALARM_INDEX_EVERYTHING;
				BA_WriteConfig(NEXT_INDEX, PLC_BA_config_index, PLC_BA_config_mask);
				substatus := 1;
			elsif PLC_BA_command = ALARM_COMMAND_DISABLE then
				NEXT_STATUS := ALARM_STATUS_OFF;
				NEXT_INDEX := ALARM_INDEX_NOTHING;
				BA_WriteConfig(NEXT_INDEX, PLC_BA_config_index, PLC_BA_config_mask);
				substatus := 1;
			elsif PLC_BA_command = ALARM_COMMAND_ENABLE then
				NEXT_STATUS := ALARM_STATUS_ENABLED;
				substatus := 2;
			elsif PLC_BA_command = ALARM_COMMAND_TEST then
				NEXT_STATUS := ALARM_STATUS_TESTING;
				substatus := 2;
			elsif BA_CheckSensors(PLC_BA_config_index) then
				substatus := 2;
			else
				substatus := 2;
			end_if;

		ALARM_STATUS_ENABLED:
			if PLC_BA_command = ALARM_COMMAND_DISABLE then
				NEXT_STATUS := ALARM_STATUS_OFF;
				NEXT_INDEX := ALARM_INDEX_NOTHING;
				BA_WriteConfig(NEXT_INDEX, PLC_BA_config_index, PLC_BA_config_mask);
				substatus := 1;
			elsif PLC_BA_command = ALARM_COMMAND_TEST then
				NEXT_STATUS := ALARM_STATUS_TESTING;
				substatus := 2;
			elsif BA_CheckSensors(PLC_BA_config_index) then
				substatus := 2;
			else
				NEXT_STATUS := ALARM_STATUS_RINGING;
				substatus := 2;
			end_if;

		ALARM_STATUS_RINGING:
			if PLC_BA_command = ALARM_COMMAND_ACK then
				NEXT_STATUS := ALARM_STATUS_MUTED;
				substatus := 2;
			elsif PLC_BA_command = ALARM_COMMAND_TEST then
				NEXT_STATUS := ALARM_STATUS_TESTING;
				substatus := 2;
			elsif BA_CheckSensors(PLC_BA_config_index) then
				substatus := 2;
			else
				NEXT_STATUS := ALARM_STATUS_RINGING;
				substatus := 2;
			end_if;

		ALARM_STATUS_MUTED:
			if PLC_BA_command = ALARM_COMMAND_DISABLE then
				NEXT_STATUS := ALARM_STATUS_OFF;
				NEXT_INDEX := ALARM_INDEX_NOTHING;
				BA_WriteConfig(NEXT_INDEX, PLC_BA_config_index, PLC_BA_config_mask);
				substatus := 1;
			elsif PLC_BA_command = ALARM_COMMAND_TEST then
				NEXT_STATUS := ALARM_STATUS_TESTING;
				substatus := 2;
			elsif BA_CheckSensors(PLC_BA_config_index) then
				substatus := 2;
			else
				substatus := 2;
			end_if;

		ALARM_STATUS_TESTING:
			if PLC_BA_command = ALARM_COMMAND_DISABLE then
				NEXT_STATUS := ALARM_STATUS_OFF;
				NEXT_INDEX := ALARM_INDEX_NOTHING;
				BA_WriteConfig(NEXT_INDEX, PLC_BA_config_index, PLC_BA_config_mask);
				substatus := 1;
			else
				BA_TestConfig();
				substatus := 1;
			end_if;

		else
			BA_ClearOKs();
			NEXT_INDEX := ALARM_INDEX_NOTHING;
			NEXT_STATUS := ALARM_STATUS_OFF;
			BA_WriteConfig(NEXT_INDEX, PLC_BA_config_index, PLC_BA_config_mask);
			substatus := 1;
		end_case;

		(* NB: only here !! *)
		if PLC_BA_command <> ALARM_COMMAND_NONE then
			SRV_BA_command := ALARM_COMMAND_NONE;
		end_if;

	else (* ------------------------------------------------------------- *)
		substatus := 0;

	end_case;

	BA_WriteLeds(NEXT_INDEX, NEXT_STATUS);
	if PLC_BA_status <> NEXT_STATUS then
		PLC_BA_status  := NEXT_STATUS;
		if NEXT_STATUS = ALARM_STATUS_RINGING then
			if not PLC_BA_ringing_flag then PLC_BA_ringing_flag := true; end_if;
		else
			if PLC_BA_ringing_flag then PLC_BA_ringing_flag := false; end_if;
		end_if;

	end_if;

END_PROGRAM

(* ---- Buzzer.st ---- *)
(****************************************************************************
**
** Copyright (C) 2021 Francesco Mandracci
** Contact: https://github.com/fmandracci/smart-home
**
** This file is part of the Smart Home Framework.
**
** Commercial License Usage
** Licensees holding valid commercial licenses may use this file in
** accordance with the terms contained in a written agreement
** between you and the copyright owner.
**
** GNU Lesser General Public License Usage
** Alternatively, this file may be used under the terms of the GNU Lesser
** General Public License version 3 as published by the Free Software
** Foundation and appearing in the file LICENSE included in the
** packaging of this file. Please review the following information to
** ensure the GNU Lesser General Public License version 3 requirements
** will be met: https://www.gnu.org/licenses/lgpl-3.0.html.
**
****************************************************************************)

PROGRAM Buzzer
#import "Crosstable.gvl"
#import "Resource1.gvl"
CONST
	QUIET_status       : UINT  := 0;
	QUIET_sound        : UDINT := 16#00000000;
	QUIET_period       : TIME  := T#2000ms;

	ONE_ALARM_status   : UINT  := 1;
	ONE_ALARM_sound    : UDINT := 16#03193264; (* count=3; off=0.25s; on=0.50s; volume=100%; total=2.25s *)
	ONE_ALARM_period   : TIME  := T#3000ms;

	BOTH_ALARMS_status : UINT  := 2;
	BOTH_ALARMS_sound  : UDINT := 16#03193264; (* count=6; off=0.25s; on=0.50s; volume=100%; total=4.50s *)
	BOTH_ALARMS_period : TIME  := T#5000ms;

	ONE_TIMER_status   : UINT  := 3;
	ONE_TIMER_sound    : UDINT := 16#03030364; (* count=3; off=0.03s; on=0.03s; volume=100%; total=0.18s *)
	ONE_TIMER_period   : TIME  :=  T#500ms;

	BOTH_TIMERS_status : UINT  := 4;
	BOTH_TIMERS_sound  : UDINT := 16#06030364; (* count=6; off=0.03s; on=0.03s; volume=100%; total=0.36s *)
	BOTH_TIMERS_period : TIME  :=  T#500ms;
END_CONST
VAR
	status : UINT := QUIET_status;
	sound : UDINT := QUIET_sound;
	period : TIME := QUIET_period;
	next_status : UINT := QUIET_status;
	timer : TON;
END_VAR;

	(* retrieve alarm status from Burglar Alarm *)
	case PLC_BA_status of
    ALARM_STATUS_ZERO,
    ALARM_STATUS_OFF,
    ALARM_STATUS_ARMED,
    ALARM_STATUS_ENABLED:
        PLC_buzzer_alarm := false;
    ALARM_STATUS_RINGING:
        PLC_buzzer_alarm := true;
    ALARM_STATUS_MUTED,
    ALARM_STATUS_TESTING:
        PLC_buzzer_alarm := false;
    else
        ;
	end_case;

	(* retrieving blackout status from both Electric Panel and Burglar Alarm *)
	PLC_buzzer_blackout_or_overload := PLC_EP_BlackoutDetected or PLC_BA_BlackoutDetected or PLC_EP_OverloadDetected; (* vedi TcpUpdate.st *)

	(* timer values are always from the local hmi *)

	(* buzzer state machine: conditions *)
	if PLC_buzzer_alarm and PLC_buzzer_blackout_or_overload then
		next_status := BOTH_ALARMS_status;
		sound := BOTH_ALARMS_sound;
		period := BOTH_ALARMS_period;
	elsif PLC_buzzer_alarm or PLC_buzzer_blackout_or_overload then
		next_status := ONE_ALARM_status;
		sound := ONE_ALARM_sound;
		period := ONE_ALARM_period;
	elsif PLC_buzzer_timer_1 and PLC_buzzer_timer_2 then
		next_status := BOTH_TIMERS_status;
		sound := BOTH_TIMERS_sound;
		period := BOTH_TIMERS_period;
	elsif PLC_buzzer_timer_1 or PLC_buzzer_timer_2 then
		next_status := ONE_TIMER_status;
		sound := ONE_TIMER_sound;
		period := ONE_TIMER_period;
	else
		next_status := QUIET_status;
		sound := QUIET_sound;
		period := QUIET_period;
	end_if;

	(* buzzer state machine: actions *)
	if status <> next_status then
		(* entering new buzzer status *)
		status := next_status;
		PLC_BUZZER := sound; (* <-----= first buzzer *)
		timer(IN := FALSE);
	else
		(* same buzzer status *)
		timer(IN := TRUE, PT := period );
		if timer.Q then
			PLC_BUZZER := sound; (* <-----= buzzer repeat *)
			timer(IN := FALSE);
		end_if;
	end_if;

END_PROGRAM

(* ---- EP_LoadBalancer.st ---- *)
(****************************************************************************
**
** Copyright (C) 2021 Francesco Mandracci
** Contact: https://github.com/fmandracci/smart-home
**
** This file is part of the Smart Home Framework.
**
** Commercial License Usage
** Licensees holding valid commercial licenses may use this file in
** accordance with the terms contained in a written agreement
** between you and the copyright owner.
**
** GNU Lesser General Public License Usage
** Alternatively, this file may be used under the terms of the GNU Lesser
** General Public License version 3 as published by the Free Software
** Foundation and appearing in the file LICENSE included in the
** packaging of this file. Please review the following information to
** ensure the GNU Lesser General Public License version 3 requirements
** will be met: https://www.gnu.org/licenses/lgpl-3.0.html.
**
****************************************************************************)

PROGRAM EP_LoadBalancer
#import "Crosstable.gvl"
#import "Resource1.gvl"
VAR
	last_assigned : UINT := 0;
	first_refused : UINT := 0;
	i: UINT;
	base: UINT;
	total_requested_W: UINT;
	total_assigned_W: UINT;
	tic_in_tac: UINT := 0;
END_VAR

	tic_in_tac := (tic_in_tac + 1) mod TacPeriod_s;

	if PLC_Tn_count > 0 then

		if (tic_in_tac = Decision_TicInTac) then (* the decision time has come ! *)
			total_requested_W := 0;
			total_assigned_W := 0;

			if first_refused = 0 then
				base := last_assigned;     (* i.e. we start from the next one *)
			elsif first_refused = 1 then
				base := 6;                 (* i.e. we start from the first_refused *)
				first_refused := 0;
			else
				base := first_refused - 1; (* i.e. we start from the first_refused *)
				first_refused := 0;
			end_if;

			for i := 0 to 5 by 1 do
				case (((base + i) mod 6) + 1) of
				1: EP_ManageRequest(1, PLC_T1_requested_W, PLC_EP_T1_assigned_W, total_requested_W, total_assigned_W, last_assigned, first_refused);
				2: EP_ManageRequest(2, PLC_T2_requested_W, PLC_EP_T2_assigned_W, total_requested_W, total_assigned_W, last_assigned, first_refused);
				3: EP_ManageRequest(3, PLC_T3_requested_W, PLC_EP_T3_assigned_W, total_requested_W, total_assigned_W, last_assigned, first_refused);
				4: EP_ManageRequest(4, PLC_T4_requested_W, PLC_EP_T4_assigned_W, total_requested_W, total_assigned_W, last_assigned, first_refused);
				5: EP_ManageRequest(5, PLC_T5_requested_W, PLC_EP_T5_assigned_W, total_requested_W, total_assigned_W, last_assigned, first_refused);
				6: EP_ManageRequest(6, PLC_T6_requested_W, PLC_EP_T6_assigned_W, total_requested_W, total_assigned_W, last_assigned, first_refused);
				else ;
				end_case;
	 	    end_for;

			PLC_EP_requested_W := total_requested_W;
			PLC_EP_assigned_W := total_assigned_W;

	    end_if;

	else
		if PLC_EP_T1_assigned_W <> 0 then PLC_EP_T1_assigned_W := 0; end_if;
		if PLC_EP_T2_assigned_W <> 0 then PLC_EP_T2_assigned_W := 0; end_if;
		if PLC_EP_T3_assigned_W <> 0 then PLC_EP_T3_assigned_W := 0; end_if;
		if PLC_EP_T4_assigned_W <> 0 then PLC_EP_T4_assigned_W := 0; end_if;
		if PLC_EP_T5_assigned_W <> 0 then PLC_EP_T5_assigned_W := 0; end_if;
		if PLC_EP_T6_assigned_W <> 0 then PLC_EP_T6_assigned_W := 0; end_if;

		if PLC_EP_requested_W <> 0 then PLC_EP_requested_W := 0; end_if;
		if PLC_EP_assigned_W <> 0 then PLC_EP_assigned_W := 0; end_if;

	end_if;

	PLC_EP_tic_in_tac := tic_in_tac;

END_PROGRAM

(* ---- EP_Relays.st ---- *)
(****************************************************************************
**
** Copyright (C) 2021 Francesco Mandracci
** Contact: https://github.com/fmandracci/smart-home
**
** This file is part of the Smart Home Framework.
**
** Commercial License Usage
** Licensees holding valid commercial licenses may use this file in
** accordance with the terms contained in a written agreement
** between you and the copyright owner.
**
** GNU Lesser General Public License Usage
** Alternatively, this file may be used under the terms of the GNU Lesser
** General Public License version 3 as published by the Free Software
** Foundation and appearing in the file LICENSE included in the
** packaging of this file. Please review the following information to
** ensure the GNU Lesser General Public License version 3 requirements
** will be met: https://www.gnu.org/licenses/lgpl-3.0.html.
**
****************************************************************************)

PROGRAM EP_Relays
#import "Crosstable.gvl"
#import "Resource1.gvl"
VAR
	n : UINT := 0;
END_VAR;

    if not PLC_Iam_EP then
		return;
	end_if;

	if PLC_EP_enabled_relays > 0 then
		(* normally open relays, custom logic *)

		if PLC_EP_enabled_relays >= 1 then EP_SetDigOut_relay(1, PLC_EP_relay_A); end_if;
		if PLC_EP_enabled_relays >= 2 then EP_SetDigOut_relay(2, PLC_EP_relay_B); end_if;
		if PLC_EP_enabled_relays >= 3 then EP_SetDigOut_relay(3, PLC_EP_relay_C); end_if;
		if PLC_EP_enabled_relays >= 4 then EP_SetDigOut_relay(4, PLC_EP_relay_D); end_if;

		if PLC_EP_enabled_relays >= 5 then EP_SetDigOut_relay(5, PLC_EP_relay_E); end_if;
		if PLC_EP_enabled_relays >= 6 then EP_SetDigOut_relay(6, PLC_EP_relay_F); end_if;
		if PLC_EP_enabled_relays >= 7 then EP_SetDigOut_relay(7, PLC_EP_relay_G); end_if;
		if PLC_EP_enabled_relays >= 8 then EP_SetDigOut_relay(8, PLC_EP_relay_H); end_if;

	elsif PLC_EP_enabled_relays < 0 then
		(* normally closed relays, overload cutoff and manual rearm *)

	    if PLC_EP_OverloadDetected then
			(* overload cutoff (each n seconds) *)
			if n < 4 then
				n := n + 1;
			else
				n := 0;
				if    PLC_EP_enabled_relays <= -8 and not PLC_EP_relay_H then PLC_EP_relay_H := true; EP_SetDigOut_relay(8, true);
				elsif PLC_EP_enabled_relays <= -7 and not PLC_EP_relay_G then PLC_EP_relay_G := true; EP_SetDigOut_relay(7, true);
				elsif PLC_EP_enabled_relays <= -6 and not PLC_EP_relay_F then PLC_EP_relay_F := true; EP_SetDigOut_relay(6, true);
				elsif PLC_EP_enabled_relays <= -5 and not PLC_EP_relay_E then PLC_EP_relay_E := true; EP_SetDigOut_relay(5, true);

				elsif PLC_EP_enabled_relays <= -4 and not PLC_EP_relay_D then PLC_EP_relay_D := true; EP_SetDigOut_relay(4, true);
				elsif PLC_EP_enabled_relays <= -3 and not PLC_EP_relay_C then PLC_EP_relay_C := true; EP_SetDigOut_relay(3, true);
				elsif PLC_EP_enabled_relays <= -2 and not PLC_EP_relay_B then PLC_EP_relay_B := true; EP_SetDigOut_relay(2, true);
				elsif PLC_EP_enabled_relays <= -1 and not PLC_EP_relay_A then PLC_EP_relay_A := true; EP_SetDigOut_relay(1, true);
				end_if;
		    end_if;
		else
			(* manual rearm *)
			n:= 0;
			if PLC_EP_enabled_relays <= -1 then EP_SetDigOut_relay(1, PLC_EP_relay_A); end_if;
			if PLC_EP_enabled_relays <= -2 then EP_SetDigOut_relay(2, PLC_EP_relay_B); end_if;
			if PLC_EP_enabled_relays <= -3 then EP_SetDigOut_relay(3, PLC_EP_relay_C); end_if;
			if PLC_EP_enabled_relays <= -4 then EP_SetDigOut_relay(4, PLC_EP_relay_D); end_if;

			if PLC_EP_enabled_relays <= -5 then EP_SetDigOut_relay(5, PLC_EP_relay_E); end_if;
			if PLC_EP_enabled_relays <= -6 then EP_SetDigOut_relay(6, PLC_EP_relay_F); end_if;
			if PLC_EP_enabled_relays <= -7 then EP_SetDigOut_relay(7, PLC_EP_relay_G); end_if;
			if PLC_EP_enabled_relays <= -8 then EP_SetDigOut_relay(8, PLC_EP_relay_H); end_if;
		end_if;
	end_if;

END_PROGRAM

(* ---- EP_Wattmeters.st ---- *)
(****************************************************************************
**
** Copyright (C) 2021 Francesco Mandracci
** Contact: https://github.com/fmandracci/smart-home
**
** This file is part of the Smart Home Framework.
**
** Commercial License Usage
** Licensees holding valid commercial licenses may use this file in
** accordance with the terms contained in a written agreement
** between you and the copyright owner.
**
** GNU Lesser General Public License Usage
** Alternatively, this file may be used under the terms of the GNU Lesser
** General Public License version 3 as published by the Free Software
** Foundation and appearing in the file LICENSE included in the
** packaging of this file. Please review the following information to
** ensure the GNU Lesser General Public License version 3 requirements
** will be met: https://www.gnu.org/licenses/lgpl-3.0.html.
**
****************************************************************************)

PROGRAM EP_Wattmeters
#import "Crosstable.gvl"
#import "Resource1.gvl"
VAR
	timer_blackout : TON;
	mask : UINT;
END_VAR;

    if not PLC_Iam_EP then
		return;
	end_if;

	(* --------------------- each second --------------------- *)

	mask := 0;

    if PLC_EP_enabled_wattmeters >= 1 then
		if (PLC_control_type = ControlType_6 and NODE_32_STATUS = NODE_NODE_OK) or (PLC_control_type <> ControlType_6 and NODE_15_STATUS = NODE_NODE_OK) then
			mask := mask + 1;
			EP_WattmeterFull(1, PLC_EP_wattmeter_M_W, PLC_EP_wattmeter_M_var, PLC_EP_wattmeter_M_VA,
			                 PLC_EP_wattmeter_M_pf, PLC_EP_wattmeter_M_Hz, PLC_EP_wattmeter_M_V,
							 PLC_EP_wattmeter_M_1_A, PLC_EP_wattmeter_M_2_A, PLC_EP_wattmeter_M_3_A, PLC_EP_wattmeter_M_A,
							 PLC_EP_wattmeter_M_kWh, PLC_EP_wattmeter_M_e_kWh);

			(* ------- blackout detection ------- *)
			if BlackoutDetected_enable then
				if PLC_EP_blackout_flag then
					(* NB: no delay *)
					PLC_EP_blackout_flag := false; (* --> falling PLC_EP_BlackoutDetected Alarm *)
					timer_blackout(IN := FALSE);
				end_if;
			end_if;

			(* ------- overload detection ------- *)
			if (PLC_EP_overload_W > 0) and (PLC_EP_wattmeter_M_W > UINT_TO_INT(PLC_EP_overload_W)) then
				PLC_EP_overload_flag := true; (* --> rising PLC_EP_OverloadDetected Alarm *)
			else
				if PLC_EP_overload_flag then PLC_EP_overload_flag := false; end_if; (* NB: avoid useless alarm checking in the plc engine *)
			end_if;

		else
			(* ------- blackout detection ------- *)
			if BlackoutDetected_enable then
				timer_blackout(IN := TRUE, PT := BlackoutDetected_delay);
				if timer_blackout.Q then
					timer_blackout(IN := FALSE);
					PLC_EP_blackout_flag := true; (* --> rising PLC_EP_BlackoutDetected Alarm *)
					(* ------- overload detection ------- *)
					if PLC_EP_overload_flag then PLC_EP_overload_flag := false; end_if; (* NB: avoid useless alarm checking in the plc engine *)
				end_if;
			end_if;

		end_if;
    end_if;

    if PLC_EP_enabled_wattmeters >= 2 then
		if (PLC_control_type = ControlType_6 and NODE_33_STATUS = NODE_NODE_OK) or (PLC_control_type <> ControlType_6 and NODE_16_STATUS = NODE_NODE_OK)  then
			mask := mask + 2;
			EP_WattmeterFull(2, PLC_EP_wattmeter_F_W, PLC_EP_wattmeter_F_var, PLC_EP_wattmeter_F_VA,
			                 PLC_EP_wattmeter_F_pf, PLC_EP_wattmeter_F_Hz, PLC_EP_wattmeter_F_V,
							 PLC_EP_wattmeter_F_1_A, PLC_EP_wattmeter_F_2_A, PLC_EP_wattmeter_F_3_A, PLC_EP_wattmeter_F_A,
							 PLC_EP_wattmeter_F_kWh, PLC_EP_wattmeter_F_e_kWh);
	    else
			; (* TODO: timer? *)
		end_if;
    end_if;

    if PLC_EP_enabled_wattmeters >= 3 then
		if (PLC_control_type = ControlType_6 and NODE_34_STATUS = NODE_NODE_OK) or (PLC_control_type <> ControlType_6 and NODE_17_STATUS = NODE_NODE_OK)  then
			mask := mask + 4;
			EP_Wattmeter(3, PLC_EP_wattmeter01_W, PLC_EP_wattmeter01_var, PLC_EP_wattmeter01_VA,
						PLC_EP_wattmeter01_kWh);
	    else
			; (* TODO: timer? *)
		end_if;
    end_if;

    if PLC_EP_enabled_wattmeters >= 4 then
		if (PLC_control_type = ControlType_6 and NODE_35_STATUS = NODE_NODE_OK) or (PLC_control_type <> ControlType_6 and NODE_18_STATUS = NODE_NODE_OK)  then
			mask := mask + 8;
			EP_Wattmeter(4, PLC_EP_wattmeter02_W, PLC_EP_wattmeter02_var, PLC_EP_wattmeter02_VA,
						PLC_EP_wattmeter02_kWh);
	    else
			; (* TODO: timer? *)
		end_if;
    end_if;

    if PLC_EP_enabled_wattmeters >= 5 then
		if (PLC_control_type = ControlType_6 and NODE_36_STATUS = NODE_NODE_OK) or (PLC_control_type <> ControlType_6 and NODE_19_STATUS = NODE_NODE_OK)  then
			mask := mask + 16;
			EP_Wattmeter(5, PLC_EP_wattmeter03_W, PLC_EP_wattmeter03_var, PLC_EP_wattmeter03_VA,
						 PLC_EP_wattmeter03_kWh);
	    else
			; (* TODO: timer? *)
		end_if;
    end_if;

    if PLC_EP_enabled_wattmeters >= 6 then
		if (PLC_control_type = ControlType_6 and NODE_37_STATUS = NODE_NODE_OK) or (PLC_control_type <> ControlType_6 and NODE_20_STATUS = NODE_NODE_OK)  then
			mask := mask + 32;
			EP_Wattmeter(6, PLC_EP_wattmeter04_W, PLC_EP_wattmeter04_var, PLC_EP_wattmeter04_VA,
						 PLC_EP_wattmeter04_kWh);
	    else
			; (* TODO: timer? *)
		end_if;
    end_if;

    if PLC_EP_enabled_wattmeters >= 7 then
		if (PLC_control_type = ControlType_6 and NODE_38_STATUS = NODE_NODE_OK) or (PLC_control_type <> ControlType_6 and NODE_21_STATUS = NODE_NODE_OK)  then
			mask := mask + 64;
			EP_Wattmeter(7, PLC_EP_wattmeter05_W, PLC_EP_wattmeter05_var, PLC_EP_wattmeter05_VA,
						 PLC_EP_wattmeter05_kWh);
	    else
			; (* TODO: timer? *)
		end_if;
    end_if;

    if PLC_EP_enabled_wattmeters >= 8 then
		if (PLC_control_type = ControlType_6 and NODE_39_STATUS = NODE_NODE_OK) or (PLC_control_type <> ControlType_6 and NODE_22_STATUS = NODE_NODE_OK)  then
			mask := mask + 128;
			EP_Wattmeter(8, PLC_EP_wattmeter06_W, PLC_EP_wattmeter06_var, PLC_EP_wattmeter06_VA,
						 PLC_EP_wattmeter06_kWh);
	    else
			; (* TODO: timer? *)
		end_if;
    end_if;

    if PLC_EP_enabled_wattmeters >= 9 then
		if (PLC_control_type = ControlType_6 and NODE_40_STATUS = NODE_NODE_OK) or (PLC_control_type <> ControlType_6 and NODE_23_STATUS = NODE_NODE_OK)  then
			mask := mask + 256;
			EP_Wattmeter(9, PLC_EP_wattmeter07_W, PLC_EP_wattmeter07_var, PLC_EP_wattmeter07_VA,
						 PLC_EP_wattmeter07_kWh);
	    else
			; (* TODO: timer? *)
		end_if;
    end_if;

    if PLC_EP_enabled_wattmeters >= 10 then
		if (PLC_control_type = ControlType_6 and NODE_41_STATUS = NODE_NODE_OK) or (PLC_control_type <> ControlType_6 and NODE_24_STATUS = NODE_NODE_OK)  then
			mask := mask + 512;
			EP_Wattmeter(10, PLC_EP_wattmeter08_W, PLC_EP_wattmeter08_var, PLC_EP_wattmeter08_VA,
						 PLC_EP_wattmeter08_kWh);
	    else
			; (* TODO: timer? *)
		end_if;
    end_if;

    if PLC_EP_enabled_wattmeters >= 11 then
		if (PLC_control_type = ControlType_6 and NODE_42_STATUS = NODE_NODE_OK) or (PLC_control_type <> ControlType_6 and NODE_25_STATUS = NODE_NODE_OK)  then
			mask := mask + 1024;
			EP_Wattmeter(11, PLC_EP_wattmeter09_W, PLC_EP_wattmeter09_var, PLC_EP_wattmeter09_VA,
						 PLC_EP_wattmeter09_kWh);
	    else
			; (* TODO: timer? *)
		end_if;
    end_if;

    if PLC_EP_enabled_wattmeters >= 12 then
		if (PLC_control_type = ControlType_6 and NODE_43_STATUS = NODE_NODE_OK) or (PLC_control_type <> ControlType_6 and NODE_26_STATUS = NODE_NODE_OK)  then
			mask := mask + 2048;
			EP_Wattmeter(12, PLC_EP_wattmeter10_W, PLC_EP_wattmeter10_var, PLC_EP_wattmeter10_VA,
						 PLC_EP_wattmeter10_kWh);
	    else
			; (* TODO: timer? *)
		end_if;
    end_if;

	PLC_EP_wattmeters_ok := mask;

END_PROGRAM

(* ---- Events.st ---- *)
(****************************************************************************
**
** Copyright (C) 2021 Francesco Mandracci
** Contact: https://github.com/fmandracci/smart-home
**
** This file is part of the Smart Home Framework.
**
** Commercial License Usage
** Licensees holding valid commercial licenses may use this file in
** accordance with the terms contained in a written agreement
** between you and the copyright owner.
**
** GNU Lesser General Public License Usage
** Alternatively, this file may be used under the terms of the GNU Lesser
** General Public License version 3 as published by the Free Software
** Foundation and appearing in the file LICENSE included in the
** packaging of this file. Please review the following information to
** ensure the GNU Lesser General Public License version 3 requirements
** will be met: https://www.gnu.org/licenses/lgpl-3.0.html.
**
****************************************************************************)

PROGRAM Events
#import "Crosstable.gvl"
#import "Resource1.gvl"
VAR

END_VAR

;

END_PROGRAM

(* ---- Init.st ---- *)
(****************************************************************************
**
** Copyright (C) 2021 Francesco Mandracci
** Contact: https://github.com/fmandracci/smart-home
**
** This file is part of the Smart Home Framework.
**
** Commercial License Usage
** Licensees holding valid commercial licenses may use this file in
** accordance with the terms contained in a written agreement
** between you and the copyright owner.
**
** GNU Lesser General Public License Usage
** Alternatively, this file may be used under the terms of the GNU Lesser
** General Public License version 3 as published by the Free Software
** Foundation and appearing in the file LICENSE included in the
** packaging of this file. Please review the following information to
** ensure the GNU Lesser General Public License version 3 requirements
** will be met: https://www.gnu.org/licenses/lgpl-3.0.html.
**
****************************************************************************)

PROGRAM Init
#import "Crosstable.gvl"
#import "Resource1.gvl"

	PLC_PLC_Version := 1200;

	(* Fast I/O on TPX1043_03_C only *)
	if PLC_PRODUCT_ID = 16#1043030C then
	    PLC_FastIO_Ena := 16#000000FF;
	    PLC_FastIO_Dir := 16#000000F0;
	end_if;

	(* NB: in hmi.ini: disable_all_nodes=true *)

	if Vbase_Ventola < 100 then Vbase_Ventola := 100; end_if;

	(* TCP0..TCP7 *)
	if (PLC_EP_exists     and not PLC_Iam_EP) then NODE_01_STATUS := 1; end_if;
	if (PLC_Tn_count >= 1 and not PLC_Iam_T1) then NODE_02_STATUS := 1; end_if;
	if (PLC_Tn_count >= 2 and not PLC_Iam_T2) then NODE_03_STATUS := 1; end_if;
	if (PLC_Tn_count >= 3 and not PLC_Iam_T3) then NODE_04_STATUS := 1; end_if;
	if (PLC_Tn_count >= 4 and not PLC_Iam_T4) then NODE_05_STATUS := 1; end_if;
	if (PLC_Tn_count >= 5 and not PLC_Iam_T5) then NODE_06_STATUS := 1; end_if;
	if (PLC_Tn_count >= 6 and not PLC_Iam_T6) then NODE_07_STATUS := 1; end_if;
	if (PLC_BA_exists     and not PLC_Iam_BA) then NODE_08_STATUS := 1; end_if;

    if (PLC_Iam_EP or PLC_Iam_T1 or PLC_Iam_T2 or PLC_Iam_T3 or PLC_Iam_T4 or PLC_Iam_T5 or PLC_Iam_T6 or PLC_Iam_BA) then
		(* TCPS *)
		NODE_09_STATUS := 1;
	end_if;

	if PLC_Iam_EP then (* --------------------------------------------------------- *)

		(* INPUT: wattmeters *)
		if PLC_EP_enabled_wattmeters >= 1 then
			if PLC_control_type = ControlType_1 or PLC_control_type = ControlType_7 or PLC_control_type = ControlType_12 or PLC_control_type = ControlType_13 or PLC_control_type = ControlType_14 or PLC_control_type = ControlType_15 then
				(* Finder 7M.24/7M.38 wattmeters 1..12 on RTU0 *)
				if PLC_EP_enabled_wattmeters >=  1 then NODE_15_STATUS := 1; end_if;
				if PLC_EP_enabled_wattmeters >=  2 then NODE_16_STATUS := 1; end_if;
				if PLC_EP_enabled_wattmeters >=  3 then NODE_17_STATUS := 1; end_if;
				if PLC_EP_enabled_wattmeters >=  4 then NODE_18_STATUS := 1; end_if;
				if PLC_EP_enabled_wattmeters >=  5 then NODE_19_STATUS := 1; end_if;
				if PLC_EP_enabled_wattmeters >=  6 then NODE_20_STATUS := 1; end_if;
				if PLC_EP_enabled_wattmeters >=  7 then NODE_21_STATUS := 1; end_if;
				if PLC_EP_enabled_wattmeters >=  8 then NODE_22_STATUS := 1; end_if;
				if PLC_EP_enabled_wattmeters >=  9 then NODE_23_STATUS := 1; end_if;
				if PLC_EP_enabled_wattmeters >= 10 then NODE_24_STATUS := 1; end_if;
				if PLC_EP_enabled_wattmeters >= 11 then NODE_25_STATUS := 1; end_if;
				if PLC_EP_enabled_wattmeters >= 12 then NODE_26_STATUS := 1; end_if;
			elsif PLC_control_type = ControlType_6 then
				(* Finder 7E.64 wattmeters 1..12 on RTU0 *)
				if PLC_EP_enabled_wattmeters >=  1 then NODE_32_STATUS := 1; end_if;
				if PLC_EP_enabled_wattmeters >=  2 then NODE_33_STATUS := 1; end_if;
				if PLC_EP_enabled_wattmeters >=  3 then NODE_34_STATUS := 1; end_if;
				if PLC_EP_enabled_wattmeters >=  4 then NODE_35_STATUS := 1; end_if;
				if PLC_EP_enabled_wattmeters >=  5 then NODE_36_STATUS := 1; end_if;
				if PLC_EP_enabled_wattmeters >=  6 then NODE_37_STATUS := 1; end_if;
				if PLC_EP_enabled_wattmeters >=  7 then NODE_38_STATUS := 1; end_if;
				if PLC_EP_enabled_wattmeters >=  8 then NODE_39_STATUS := 1; end_if;
				if PLC_EP_enabled_wattmeters >=  9 then NODE_40_STATUS := 1; end_if;
				if PLC_EP_enabled_wattmeters >= 10 then NODE_41_STATUS := 1; end_if;
				if PLC_EP_enabled_wattmeters >= 11 then NODE_42_STATUS := 1; end_if;
				if PLC_EP_enabled_wattmeters >= 12 then NODE_43_STATUS := 1; end_if;
			end_if;
		end_if;

		(* OUTPUT: relays *)
		if abs(PLC_EP_enabled_relays) >= 1 then
			if PLC_control_type = ControlType_1 then
				if PLC_PRODUCT_ID = 16#1043030C then
					(* Fast I/O on GPIO *);
				elsif PLC_PRODUCT_ID = 16#100704AD or PLC_PRODUCT_ID = 16#100704AE or PLC_PRODUCT_ID = 16#100704AA or PLC_PRODUCT_ID = 16#100704AC then
					(* TPAC1007_04_AD/E/A/C Local I/O on RTU3 *)
					NODE_31_STATUS := 1;
				else
					; (* TP.. *)
				end_if;
			elsif PLC_control_type = ControlType_7 then
				(* Fast I/O on GPIO *);
			elsif PLC_control_type = ControlType_12 then
				(* Fast I/O on GPIO *);
			elsif PLC_control_type = ControlType_13 then
				(* TPAC1007_04_AD Local I/O on RTU3 *)
				NODE_31_STATUS := 1;
			elsif PLC_control_type = ControlType_6 then
				(* MPNC base on RTU0 *)
				NODE_27_STATUS := 1;
			elsif PLC_control_type = ControlType_14 then
				(* MPNC DO16 "C" on RTU0 *)
				NODE_27_STATUS := 1;
			end_if;
		end_if;

	end_if;

	if PLC_Iam_T1 then (* --------------------------------------------------------- *)

		(* INPUT: sensors *)
		if PLC_control_type = ControlType_3 or PLC_control_type = ControlType_4 or PLC_control_type = ControlType_13 or PLC_control_type = ControlType_15 then
			NODE_31_STATUS := 1; (* TPAC1007_04_AD Local I/O AI1..3 on RTU3 *)
		elsif PLC_control_type = ControlType_5 or PLC_control_type = ControlType_8 or PLC_control_type = ControlType_12 then
			NODE_28_STATUS := 1; (* first (T,H) sensor on RTU3 *)
			if PLC_T1_enabled_sensors <= -2 then NODE_29_STATUS := 1; end_if; (* second (T,H) sensor on RTU3 *)
			if PLC_T1_enabled_sensors <= -3 then NODE_30_STATUS := 1; end_if; (* third (T,H) sensor on RTU3 *)
		elsif PLC_control_type = ControlType_14 or PLC_control_type = ControlType_6 then
			NODE_27_STATUS := 1; (* MPNC 4xAI4 on RTU0 *)
		elsif PLC_control_type = ControlType_7 or PLC_control_type = ControlType_10 then
			NODE_13_STATUS := 1; (* MPNE_C AI2+AO1 on RTU0 *)
		elsif PLC_control_type = ControlType_11 then
			NODE_13_STATUS := 1; (* MPNE_C AI2+AO1 on RTU0 *)
		end_if;

		(* INPUT/OUTPUT: lamps *)
		if PLC_control_type = ControlType_3 or PLC_control_type = ControlType_4 then
			NODE_31_STATUS := 1; (* TPAC1007_04_AD Local I/O DO1..5 DI7..11 on RTU3 *)
		elsif PLC_control_type = ControlType_5 or PLC_control_type = ControlType_8 then
			NODE_10_STATUS := 1; (* Fast I/O FO5..8 FI1..4 on GPIO *)
		else
			; (* no lamps *)
		end_if;

		(* OUTPUT: thermo *)
		if PLC_control_type = ControlType_3 then
			NODE_31_STATUS := 1; (* TPAC1007_04_AD Local I/O DO6 on RTU3 *)
		elsif PLC_control_type = ControlType_4 or PLC_control_type = ControlType_5 or PLC_control_type = ControlType_8 then
			NODE_10_STATUS := 1; (* ARQ01 on RTU0 *)
		elsif PLC_control_type = ControlType_6 then
			NODE_27_STATUS := 1; (* MPNC DO5..8 on RTU0 *)
		elsif PLC_control_type = ControlType_14 then
			NODE_27_STATUS := 1; (* MPNC DO1..4 on RTU0 *)
		elsif PLC_control_type = ControlType_7 or PLC_control_type = ControlType_10 then
			NODE_13_STATUS := 1; (* MPNE_C DO1..4 on RTU0 *)
		elsif PLC_control_type = ControlType_12 then
			; (* Fast I/O FO8 on GPIO *)
		elsif PLC_control_type = ControlType_13 then
			NODE_31_STATUS := 1; (* TPAC1007_04_AD Local I/O DO1..3+4 on RTU3 *)
		elsif PLC_control_type = ControlType_15 then
			NODE_31_STATUS := 1; (* TPAC1007_04_AD Local I/O DO8 on RTU3 *)
		end_if;

		(* retentives *)

		SRV_T1_temperature_setpoint := Tn_CheckSetPoint_T(PLC_T1_temperature_setpoint);
		SRV_T1_temperature_setpoint_nt := Tn_CheckSetPoint_T(PLC_T1_temperature_setpoint_nt);
		SRV_T1_humidity_setpoint := Tn_CheckSetPoint_H(PLC_T1_humidity_setpoint);
		SRV_T1_humidity_setpoint_nt := Tn_CheckSetPoint_H(PLC_T1_humidity_setpoint_nt);
		SRV_T1_heating_status := PLC_T1_heating_status;
		PLC_T1_sunrise := PLC_sunrise; PLC_T1_sunset := PLC_sunset;
		SRV_T1_sunrise := PLC_sunrise; SRV_T1_sunset := PLC_sunset;
		SRV_T1_lamp_1 := PLC_T1_lamp_1; SRV_T1_lamp_2 := PLC_T1_lamp_2; SRV_T1_lamp_3 := PLC_T1_lamp_3; SRV_T1_lamp_4 := PLC_T1_lamp_4; SRV_T1_lamp_5 := PLC_T1_lamp_5;
	end_if;

	if PLC_Iam_T2 then (* --------------------------------------------------------- *)

		(* INPUT: sensors *)
		if PLC_control_type = ControlType_3 or PLC_control_type = ControlType_4 or PLC_control_type = ControlType_13 or PLC_control_type = ControlType_15 then
			NODE_31_STATUS := 1; (* TPAC1007_04_AD Local I/O AI1..3 on RTU3 *)
		elsif PLC_control_type = ControlType_5 or PLC_control_type = ControlType_8 then
			NODE_28_STATUS := 1; (* first (T,H) sensor on RTU3 *)
			if PLC_T2_enabled_sensors <= -2 then NODE_29_STATUS := 1; end_if; (* second (T,H) sensor on RTU3 *)
			if PLC_T2_enabled_sensors <= -3 then NODE_30_STATUS := 1; end_if; (* third (T,H) sensor on RTU3 *)
		elsif PLC_control_type = ControlType_14 or PLC_control_type = ControlType_6 then
			NODE_27_STATUS := 1; (* MPNC 4xAI4 on RTU0 *)
		elsif PLC_control_type = ControlType_7 or PLC_control_type = ControlType_10 then
			NODE_13_STATUS := 1; (* MPNE_C AI2+AO1 on RTU0 *)
		elsif PLC_control_type = ControlType_11 then
			NODE_13_STATUS := 1; (* MPNE_C AI2+AO1 on RTU0 *)
		end_if;

		(* INPUT/OUTPUT: lamps *)
		if PLC_control_type = ControlType_3 or PLC_control_type = ControlType_4 then
			NODE_31_STATUS := 1; (* TPAC1007_04_AD Local I/O DO1..5 DI7..11 on RTU3 *)
		elsif PLC_control_type = ControlType_5 or PLC_control_type = ControlType_8 then
			NODE_10_STATUS := 1; (* Fast I/O FO5..8 FI1..4 on GPIO *)
		else
			; (* no lamps *)
		end_if;

		(* OUTPUT: thermo *)
		if PLC_control_type = ControlType_3 then
			NODE_31_STATUS := 1; (* TPAC1007_04_AD Local I/O DO6 on RTU3 *)
		elsif PLC_control_type = ControlType_4 or PLC_control_type = ControlType_5 or PLC_control_type = ControlType_8 then
			NODE_10_STATUS := 1; (* ARQ01 on RTU0 *)
		elsif PLC_control_type = ControlType_6 then
			NODE_27_STATUS := 1; (* MPNC DO5..8 on RTU0 *)
		elsif PLC_control_type = ControlType_14 then
			NODE_27_STATUS := 1; (* MPNC DO1..4 on RTU0 *)
		elsif PLC_control_type = ControlType_7 or PLC_control_type = ControlType_10 then
			NODE_13_STATUS := 1; (* MPNE_C DO1..4 on RTU0 *)
		elsif PLC_control_type = ControlType_13 then
			NODE_31_STATUS := 1; (* TPAC1007_04_AD Local I/O DO1..3+4 on RTU3 *)
		elsif PLC_control_type = ControlType_15 then
			NODE_31_STATUS := 1; (* TPAC1007_04_AD Local I/O DO8 on RTU3 *)
		end_if;

		(* retentives *)
		SRV_T2_temperature_setpoint := Tn_CheckSetPoint_T(PLC_T2_temperature_setpoint);
		SRV_T2_temperature_setpoint_nt := Tn_CheckSetPoint_T(PLC_T2_temperature_setpoint_nt);
		SRV_T2_humidity_setpoint := Tn_CheckSetPoint_H(PLC_T2_humidity_setpoint);
		SRV_T2_humidity_setpoint_nt := Tn_CheckSetPoint_H(PLC_T2_humidity_setpoint_nt);
		SRV_T2_heating_status := PLC_T2_heating_status;
		PLC_T2_sunrise := PLC_sunrise; PLC_T2_sunset := PLC_sunset;
		SRV_T2_sunrise := PLC_sunrise; SRV_T2_sunset := PLC_sunset;
        SRV_T2_temperature_setpoint_nt := PLC_T2_temperature_setpoint_nt; SRV_T2_humidity_setpoint_nt := PLC_T2_humidity_setpoint_nt;
        SRV_T2_lamp_1 := PLC_T2_lamp_1; SRV_T2_lamp_2 := PLC_T2_lamp_2; SRV_T2_lamp_3 := PLC_T2_lamp_3; SRV_T2_lamp_4 := PLC_T2_lamp_4; SRV_T2_lamp_5 := PLC_T2_lamp_5;
	end_if;

	if PLC_Iam_T3 then (* --------------------------------------------------------- *)

		(* INPUT: sensors *)
		if PLC_control_type = ControlType_3 or PLC_control_type = ControlType_4 or PLC_control_type = ControlType_13 or PLC_control_type = ControlType_15 then
			NODE_31_STATUS := 1; (* TPAC1007_04_AD Local I/O AI1..3 on RTU3 *)
		elsif PLC_control_type = ControlType_5 or PLC_control_type = ControlType_8 then
			NODE_28_STATUS := 1; (* first (T,H) sensor on RTU3 *)
			if PLC_T3_enabled_sensors <= -2 then NODE_29_STATUS := 1; end_if; (* second (T,H) sensor on RTU3 *)
			if PLC_T3_enabled_sensors <= -3 then NODE_30_STATUS := 1; end_if; (* third (T,H) sensor on RTU3 *)
		elsif PLC_control_type = ControlType_14 or PLC_control_type = ControlType_6 then
			NODE_27_STATUS := 1; (* MPNC 4xAI4 on RTU0 *)
		elsif PLC_control_type = ControlType_7 or PLC_control_type = ControlType_10 then
			NODE_13_STATUS := 1; (* MPNE_C AI2+AO1 on RTU0 *)
		elsif PLC_control_type = ControlType_11 then
			NODE_14_STATUS := 1; (* MPNE_D AI2+AO1 on RTU0 *)
		end_if;

		(* INPUT/OUTPUT: lamps *)
		if PLC_control_type = ControlType_3 or PLC_control_type = ControlType_4 then
			NODE_31_STATUS := 1; (* TPAC1007_04_AD Local I/O DO1..5 DI7..11 on RTU3 *)
		elsif PLC_control_type = ControlType_5 or PLC_control_type = ControlType_8 then
			NODE_10_STATUS := 1; (* Fast I/O FO5..8 FI1..4 on GPIO *)
		else
			; (* no lamps *)
		end_if;

		(* OUTPUT: thermo *)
		if PLC_control_type = ControlType_3 then
			NODE_31_STATUS := 1; (* TPAC1007_04_AD Local I/O DO6 on RTU3 *)
		elsif PLC_control_type = ControlType_4 or PLC_control_type = ControlType_5 or PLC_control_type = ControlType_8 then
			NODE_10_STATUS := 1; (* ARQ01 on RTU0 *)
		elsif PLC_control_type = ControlType_6 then
			NODE_27_STATUS := 1; (* MPNC DO5..8 on RTU0 *)
		elsif PLC_control_type = ControlType_14 then
			NODE_27_STATUS := 1; (* MPNC DO1..4 on RTU0 *)
		elsif PLC_control_type = ControlType_7 or PLC_control_type = ControlType_10 then
			NODE_13_STATUS := 1; (* MPNE_C DO1..4 on RTU0 *)
		elsif PLC_control_type = ControlType_13 then
			NODE_31_STATUS := 1; (* TPAC1007_04_AD Local I/O DO1..3+4 on RTU3 *)
		elsif PLC_control_type = ControlType_15 then
			NODE_31_STATUS := 1; (* TPAC1007_04_AD Local I/O DO8 on RTU3 *)
		end_if;

		(* retentives *)
		SRV_T3_temperature_setpoint := Tn_CheckSetPoint_T(PLC_T3_temperature_setpoint);
		SRV_T3_temperature_setpoint_nt := Tn_CheckSetPoint_T(PLC_T3_temperature_setpoint_nt);
		SRV_T3_humidity_setpoint := Tn_CheckSetPoint_H(PLC_T3_humidity_setpoint);
		SRV_T3_humidity_setpoint_nt := Tn_CheckSetPoint_H(PLC_T3_humidity_setpoint_nt);
		SRV_T3_heating_status := PLC_T3_heating_status;
		PLC_T3_sunrise := PLC_sunrise; PLC_T3_sunset := PLC_sunset;
		SRV_T3_sunrise := PLC_sunrise; SRV_T3_sunset := PLC_sunset;
        SRV_T3_temperature_setpoint_nt := PLC_T3_temperature_setpoint_nt; SRV_T3_humidity_setpoint_nt := PLC_T3_humidity_setpoint_nt;
        SRV_T3_lamp_1 := PLC_T3_lamp_1; SRV_T3_lamp_2 := PLC_T3_lamp_2; SRV_T3_lamp_3 := PLC_T3_lamp_3; SRV_T3_lamp_4 := PLC_T3_lamp_4; SRV_T3_lamp_5 := PLC_T3_lamp_5;
	end_if;

	if PLC_Iam_T4 then (* --------------------------------------------------------- *)

		(* INPUT: sensors *)
		if PLC_control_type = ControlType_3 or PLC_control_type = ControlType_4 (*or PLC_control_type = ControlType_13*) or PLC_control_type = ControlType_15 then
			NODE_31_STATUS := 1; (* TPAC1007_04_AD Local I/O AI1..3 on RTU3 *)
		elsif PLC_control_type = ControlType_5 or PLC_control_type = ControlType_8 then
			NODE_28_STATUS := 1; (* first (T,H) sensor on RTU3 *)
			if PLC_T4_enabled_sensors <= -2 then NODE_29_STATUS := 1; end_if; (* second (T,H) sensor on RTU3 *)
			if PLC_T4_enabled_sensors <= -3 then NODE_30_STATUS := 1; end_if; (* third (T,H) sensor on RTU3 *)
		elsif PLC_control_type = ControlType_6 then
			NODE_27_STATUS := 1; (* MPNC base AI1,2 on RTU0 *)
		elsif PLC_control_type = ControlType_14 or PLC_control_type = ControlType_6 then
			NODE_27_STATUS := 1; (* MPNC 4xAI4 on RTU0 *)
		elsif PLC_control_type = ControlType_7 or PLC_control_type = ControlType_10 then
			NODE_13_STATUS := 1; (* MPNE_C AI2+AO1 on RTU0 *)
		elsif PLC_control_type = ControlType_11 then
			NODE_14_STATUS := 1; (* MPNE_D AI2+AO1 on RTU0 *)
		end_if;

		(* INPUT/OUTPUT: lamps *)
		if PLC_control_type = ControlType_3 or PLC_control_type = ControlType_4 then
			NODE_31_STATUS := 1; (* TPAC1007_04_AD Local I/O DO1..5 DI7..11 on RTU3 *)
		elsif PLC_control_type = ControlType_5 or PLC_control_type = ControlType_8 then
			NODE_10_STATUS := 1; (* Fast I/O FO5..8 FI1..4 on GPIO *)
		else
			; (* no lamps *)
		end_if;

		(* OUTPUT: thermo *)
		if PLC_control_type = ControlType_3 then
			NODE_31_STATUS := 1; (* TPAC1007_04_AD Local I/O DO6 on RTU3 *)
		elsif PLC_control_type = ControlType_4 or PLC_control_type = ControlType_5 or PLC_control_type = ControlType_8 then
			NODE_10_STATUS := 1; (* ARQ01 on RTU0 *)
		elsif PLC_control_type = ControlType_6 then
			NODE_27_STATUS := 1; (* MPNC DO5..8 on RTU0 *)
		elsif PLC_control_type = ControlType_14 then
			NODE_27_STATUS := 1; (* MPNC DO1..4 on RTU0 *)
		elsif PLC_control_type = ControlType_7 or PLC_control_type = ControlType_10 then
			NODE_13_STATUS := 1; (* MPNE_C DO1..4 on RTU0 *)
		elsif PLC_control_type = ControlType_13 then
			NODE_31_STATUS := 1; (* TPAC1007_04_AD Local I/O DO1..3+4 on RTU3 *)
		elsif PLC_control_type = ControlType_15 then
			NODE_31_STATUS := 1; (* TPAC1007_04_AD Local I/O DO8 on RTU3 *)
		end_if;

		(* retentives *)
		SRV_T4_temperature_setpoint := Tn_CheckSetPoint_T(PLC_T4_temperature_setpoint);
		SRV_T4_temperature_setpoint_nt := Tn_CheckSetPoint_T(PLC_T4_temperature_setpoint_nt);
		SRV_T4_humidity_setpoint := Tn_CheckSetPoint_H(PLC_T4_humidity_setpoint);
		SRV_T4_humidity_setpoint_nt := Tn_CheckSetPoint_H(PLC_T4_humidity_setpoint_nt);
		SRV_T4_heating_status := PLC_T4_heating_status;
		PLC_T4_sunrise := PLC_sunrise; PLC_T4_sunset := PLC_sunset;
		SRV_T4_sunrise := PLC_sunrise; SRV_T4_sunset := PLC_sunset;
        SRV_T4_temperature_setpoint_nt := PLC_T4_temperature_setpoint_nt; SRV_T4_humidity_setpoint_nt := PLC_T4_humidity_setpoint_nt;
        SRV_T4_lamp_1 := PLC_T4_lamp_1; SRV_T4_lamp_2 := PLC_T4_lamp_2; SRV_T4_lamp_3 := PLC_T4_lamp_3; SRV_T4_lamp_4 := PLC_T4_lamp_4; SRV_T4_lamp_5 := PLC_T4_lamp_5;
	end_if;

	if PLC_Iam_T5 then (* --------------------------------------------------------- *)

		(* INPUT: sensors *)
		if PLC_control_type = ControlType_3 or PLC_control_type = ControlType_4 (*or PLC_control_type = ControlType_13*) or PLC_control_type = ControlType_15 then
			NODE_31_STATUS := 1; (* TPAC1007_04_AD Local I/O AI1..3 on RTU3 *)
		elsif PLC_control_type = ControlType_5 or PLC_control_type = ControlType_8 then
			NODE_28_STATUS := 1; (* first (T,H) sensor on RTU3 *)
			if PLC_T5_enabled_sensors <= -2 then NODE_29_STATUS := 1; end_if; (* second (T,H) sensor on RTU3 *)
			if PLC_T5_enabled_sensors <= -3 then NODE_30_STATUS := 1; end_if; (* third (T,H) sensor on RTU3 *)
		elsif PLC_control_type = ControlType_7 then
			NODE_28_STATUS := 1; (* first (T,H) sensor on RTU3 *)
		elsif PLC_control_type = ControlType_11 or PLC_control_type = ControlType_14 or PLC_control_type = ControlType_6 then
			; (* T1..T4 only *)
		elsif PLC_control_type = ControlType_10 then
			NODE_13_STATUS := 1; (* MPNE_C AI2+AO1 on RTU0 *)
		end_if;

		(* INPUT/OUTPUT: lamps *)
		if PLC_control_type = ControlType_3 or PLC_control_type = ControlType_4 then
			NODE_31_STATUS := 1; (* TPAC1007_04_AD Local I/O DO1..5 DI7..11 on RTU3 *)
		elsif PLC_control_type = ControlType_5 or PLC_control_type = ControlType_8 then
			NODE_10_STATUS := 1; (* Fast I/O FO5..8 FI1..4 on GPIO *)
		else
			; (* no lamps *)
		end_if;

		(* OUTPUT: thermo *)
		if PLC_control_type = ControlType_3 then
			NODE_31_STATUS := 1; (* TPAC1007_04_AD Local I/O DO6 on RTU3 *)
		elsif PLC_control_type = ControlType_4 or PLC_control_type = ControlType_5 or PLC_control_type = ControlType_8 then
			NODE_10_STATUS := 1; (* ARQ01 on RTU0 *)
		elsif PLC_control_type = ControlType_7 then
			NODE_13_STATUS := 1; (* MPNE_C DO5 on RTU0 *)
		elsif PLC_control_type = ControlType_11 or PLC_control_type = ControlType_14 or PLC_control_type = ControlType_6 then
			; (* T1..T4 only *)
		elsif PLC_control_type = ControlType_10 then
			NODE_13_STATUS := 1; (* MPNE_C DO1 on RTU0 *)
		elsif PLC_control_type = ControlType_13 then
			; (* no output *)
		elsif PLC_control_type = ControlType_15 then
			NODE_31_STATUS := 1; (* TPAC1007_04_AD Local I/O DO8 on RTU3 *)
		end_if;

		(* retentives *)
		SRV_T5_temperature_setpoint := Tn_CheckSetPoint_T(PLC_T5_temperature_setpoint);
		SRV_T5_temperature_setpoint_nt := Tn_CheckSetPoint_T(PLC_T5_temperature_setpoint_nt);
		SRV_T5_humidity_setpoint := Tn_CheckSetPoint_H(PLC_T5_humidity_setpoint);
		SRV_T5_humidity_setpoint_nt := Tn_CheckSetPoint_H(PLC_T5_humidity_setpoint_nt);
		SRV_T5_heating_status := PLC_T5_heating_status;
		PLC_T5_sunrise := PLC_sunrise; PLC_T5_sunset := PLC_sunset;
		SRV_T5_sunrise := PLC_sunrise; SRV_T5_sunset := PLC_sunset;
        SRV_T5_temperature_setpoint_nt := PLC_T5_temperature_setpoint_nt; SRV_T5_humidity_setpoint_nt := PLC_T5_humidity_setpoint_nt;
        SRV_T5_lamp_1 := PLC_T5_lamp_1; SRV_T5_lamp_2 := PLC_T5_lamp_2; SRV_T5_lamp_3 := PLC_T5_lamp_3; SRV_T5_lamp_4 := PLC_T5_lamp_4; SRV_T5_lamp_5 := PLC_T5_lamp_5;
	end_if;

	if PLC_Iam_T6 then (* --------------------------------------------------------- *)

		(* INPUT: sensors *)
		if PLC_control_type = ControlType_3 or PLC_control_type = ControlType_4 (*or PLC_control_type = ControlType_13*) or PLC_control_type = ControlType_15 then
			NODE_31_STATUS := 1; (* TPAC1007_04_AD Local I/O AI1..3 on RTU3 *)
		elsif PLC_control_type = ControlType_13 then
			; (* T1..T5 only *)
		elsif PLC_control_type = ControlType_5 or PLC_control_type = ControlType_8 then
			NODE_28_STATUS := 1; (* first (T,H) sensor on RTU3 *)
			if PLC_T6_enabled_sensors <= -2 then NODE_29_STATUS := 1; end_if; (* second (T,H) sensor on RTU3 *)
			if PLC_T6_enabled_sensors <= -3 then NODE_30_STATUS := 1; end_if; (* third (T,H) sensor on RTU3 *)
		elsif PLC_control_type = ControlType_7 then
			NODE_29_STATUS := 1; (* second (T,H) sensor on RTU3 *)
		elsif PLC_control_type = ControlType_11 or PLC_control_type = ControlType_14 or PLC_control_type = ControlType_6 then
			; (* T1..T4 only *)
		elsif PLC_control_type = ControlType_10 then
			NODE_13_STATUS := 1; (* MPNE_C AI2+AO1 on RTU0 *)
		end_if;

		(* INPUT/OUTPUT: lamps *)
		if PLC_control_type = ControlType_3 or PLC_control_type = ControlType_4 then
			NODE_31_STATUS := 1; (* TPAC1007_04_AD Local I/O DO1..5 DI7..11 on RTU3 *)
		elsif PLC_control_type = ControlType_5 or PLC_control_type = ControlType_8 then
			NODE_10_STATUS := 1; (* Fast I/O FO5..8 FI1..4 on GPIO *)
		else
			; (* no lamps *)
		end_if;

		(* OUTPUT: thermo *)
		if PLC_control_type = ControlType_3 then
			NODE_31_STATUS := 1; (* TPAC1007_04_AD Local I/O DO6 on RTU3 *)
		elsif PLC_control_type = ControlType_4 or PLC_control_type = ControlType_5 or PLC_control_type = ControlType_8 then
			NODE_10_STATUS := 1; (* ARQ01 on RTU0 *)
		elsif PLC_control_type = ControlType_7 then
			NODE_13_STATUS := 1; (* MPNE_C DO6 on RTU0 *)
		elsif PLC_control_type = ControlType_11 or PLC_control_type = ControlType_14 or PLC_control_type = ControlType_6 then
			; (* T1..T4 only *)
		elsif PLC_control_type = ControlType_10 then
			NODE_13_STATUS := 1; (* MPNE_C DO1 on RTU0 *)
		elsif PLC_control_type = ControlType_13 then
			; (* T1..T5 only *)
		elsif PLC_control_type = ControlType_15 then
			NODE_31_STATUS := 1; (* TPAC1007_04_AD Local I/O DO8 on RTU3 *)
		end_if;

		(* retentives *)
		SRV_T6_temperature_setpoint := Tn_CheckSetPoint_T(PLC_T6_temperature_setpoint);
		SRV_T6_temperature_setpoint_nt := Tn_CheckSetPoint_T(PLC_T6_temperature_setpoint_nt);
		SRV_T6_humidity_setpoint := Tn_CheckSetPoint_H(PLC_T6_humidity_setpoint);
		SRV_T6_humidity_setpoint_nt := Tn_CheckSetPoint_H(PLC_T6_humidity_setpoint_nt);
		SRV_T6_heating_status := PLC_T6_heating_status;
		PLC_T6_sunrise := PLC_sunrise; PLC_T6_sunset := PLC_sunset;
		SRV_T6_sunrise := PLC_sunrise; SRV_T6_sunset := PLC_sunset;
        SRV_T6_temperature_setpoint_nt := PLC_T6_temperature_setpoint_nt; SRV_T6_humidity_setpoint_nt := PLC_T6_humidity_setpoint_nt;
        SRV_T6_lamp_1 := PLC_T6_lamp_1; SRV_T6_lamp_2 := PLC_T6_lamp_2; SRV_T6_lamp_3 := PLC_T6_lamp_3; SRV_T6_lamp_4 := PLC_T6_lamp_4; SRV_T6_lamp_5 := PLC_T6_lamp_5;
	end_if;

    if (PLC_Iam_BA) then (* --------------------------------------------------------- *)

		PLC_BA_just_started := true;
		if PLC_BA_daytime_bitmask = 0 and PLC_BA_nighttime_bitmask = 0 and PLC_BA_everything_bitmask = 0 then
			if PLC_control_type = ControlType_6 then
				PLC_BA_daytime_bitmask := ALARM_MASK_DAYTIME_DEFAULT_6;
				PLC_BA_nighttime_bitmask := ALARM_MASK_NIGHTTIME_DEFAULT_6;
				PLC_BA_everything_bitmask := ALARM_MASK_EVERYTHING_DEFAULT_6;
			elsif PLC_control_type = ControlType_7 or PLC_control_type = ControlType_12 or PLC_control_type = ControlType_13 then
				PLC_BA_daytime_bitmask := ALARM_MASK_DAYTIME_DEFAULT_3;
				PLC_BA_nighttime_bitmask := ALARM_MASK_NIGHTTIME_DEFAULT_3;
				PLC_BA_everything_bitmask := ALARM_MASK_EVERYTHING_DEFAULT_3;
			else
				PLC_BA_daytime_bitmask := ALARM_MASK_DAYTIME_DEFAULT;
				PLC_BA_nighttime_bitmask := ALARM_MASK_NIGHTTIME_DEFAULT;
				PLC_BA_everything_bitmask := ALARM_MASK_EVERYTHING_DEFAULT;
			end_if;
		end_if;
		if PLC_BA_config_index >= ALARM_INDEX_COUNT then
			PLC_BA_config_index := ALARM_INDEX_NOTHING;
		end_if;

		if PLC_control_type = ControlType_2 then
			(* MPNE_A, MPNE_B on RTU0 *)
			if (PLC_BA_enabled_sensors >=  1) then NODE_11_STATUS := 1; end_if;
	        if (PLC_BA_enabled_sensors >= 17) then NODE_12_STATUS := 1; end_if;
			if PLC_PRODUCT_ID = 16#100704AD or PLC_PRODUCT_ID = 16#100704AE or PLC_PRODUCT_ID = 16#100704AA or PLC_PRODUCT_ID = 16#100704AC then
				(* leds and commands Local I/O on RTU3 *)
				NODE_31_STATUS := 1;
			else
				(* Fast I/O on GPIO *);
			end_if;
		elsif PLC_control_type = ControlType_7 then
			;(* Fast I/O on GPIO *)
		elsif PLC_control_type = ControlType_12 then
			;(* Fast I/O on GPIO *)
		elsif PLC_control_type = ControlType_13 then
			(* TPAC1007_04_AD Local I/O on RTU3 *)
			NODE_31_STATUS := 1;
		elsif PLC_control_type = ControlType_6 then
			(* MPNC DI16 "A,B" + DO16 "A" on RTU0 *)
			(* no leds and commands *)
			NODE_27_STATUS := 1;
		elsif PLC_control_type = ControlType_14 then
			(* MPNC DI16 "A,B" + DO16 "A,B" on RTU0 *)
			(* leds and commands on MPNC DO16 "C" *)
			NODE_27_STATUS := 1;
		end_if;

	end_if;

END_PROGRAM

(* ---- System.st ---- *)
(****************************************************************************
**
** Copyright (C) 2021 Francesco Mandracci
** Contact: https://github.com/fmandracci/smart-home
**
** This file is part of the Smart Home Framework.
**
** Commercial License Usage
** Licensees holding valid commercial licenses may use this file in
** accordance with the terms contained in a written agreement
** between you and the copyright owner.
**
** GNU Lesser General Public License Usage
** Alternatively, this file may be used under the terms of the GNU Lesser
** General Public License version 3 as published by the Free Software
** Foundation and appearing in the file LICENSE included in the
** packaging of this file. Please review the following information to
** ensure the GNU Lesser General Public License version 3 requirements
** will be met: https://www.gnu.org/licenses/lgpl-3.0.html.
**
****************************************************************************)

PROGRAM System
#import "Crosstable.gvl"
#import "Resource1.gvl"
VAR
	retval : WORD;
END_VAR

	if PLC_RELOAD_CONF then
		retval := EVT_Set(EVT_INITIALIZE);
		PLC_RELOAD_CONF := false;
		return;
	end_if;

	PLC_EP_isOK := PLC_Iam_EP or (NODE_01_STATUS = NODE_NODE_OK);
	PLC_T1_isOK := PLC_Iam_T1 or (NODE_02_STATUS = NODE_NODE_OK);
	PLC_T2_isOK := PLC_Iam_T2 or (NODE_03_STATUS = NODE_NODE_OK);
	PLC_T3_isOK := PLC_Iam_T3 or (NODE_04_STATUS = NODE_NODE_OK);
	PLC_T4_isOK := PLC_Iam_T4 or (NODE_05_STATUS = NODE_NODE_OK);
	PLC_T5_isOK := PLC_Iam_T5 or (NODE_06_STATUS = NODE_NODE_OK);
	PLC_T6_isOK := PLC_Iam_T6 or (NODE_07_STATUS = NODE_NODE_OK);
	PLC_BA_isOK := PLC_Iam_BA or (NODE_08_STATUS = NODE_NODE_OK);

	PLC_Tn_heating := (PLC_T1_heating and PLC_T1_control_type <> ControlType_15)
	               or (PLC_T2_heating and PLC_T2_control_type <> ControlType_15)
				   or (PLC_T3_heating and PLC_T3_control_type <> ControlType_15)
				   or (PLC_T4_heating and PLC_T4_control_type <> ControlType_15 and PLC_T4_control_type <> ControlType_6)
				   or (PLC_T5_heating and PLC_T5_control_type <> ControlType_15)
				   or (PLC_T6_heating and PLC_T6_control_type <> ControlType_15);

	PLC_time_bis := PLC_time + PLC_timeOffset;
	PLC_timeMin_bis := PLC_timeMin + PLC_timeOffset;
	PLC_timeMax_bis := PLC_timeMax + PLC_timeOffset;

END_PROGRAM
